LIN {X 0,Y 573.238,Z 117.075,A -85,B 0,C 180,E1 -2298.543,E2 -2298.543} C_VEL
LIN {X 0,Y 573.245,Z 117.077,A -85,B 0,C 180,E1 -2301.298,E2 -2301.298} C_VEL
LIN {X 0,Y 573.216,Z 117.081,A -85,B 0,C 180,E1 -2304.018,E2 -2304.018} C_VEL
LIN {X 0,Y 573.236,Z 117.074,A -85,B 0,C 180,E1 -2306.515,E2 -2306.515} C_VEL
LIN {X 0,Y 573.227,Z 117.08,A -85,B 0,C 180,E1 -2309.119,E2 -2309.119} C_VEL
LIN {X 0,Y 573.239,Z 117.083,A -85,B 0,C 180,E1 -2311.435,E2 -2311.435} C_VEL
LIN {X 0,Y 573.262,Z 117.073,A -85,B 0,C 180,E1 -2313.81,E2 -2313.81} C_VEL
LIN {X 0,Y 573.225,Z 117.076,A -85,B 0,C 180,E1 -2316.134,E2 -2316.134} C_VEL
LIN {X 0,Y 573.251,Z 117.082,A -85,B 0,C 180,E1 -2319.173,E2 -2319.173} C_VEL
LIN {X 0,Y 573.216,Z 117.081,A -85,B 0,C 180,E1 -2321.411,E2 -2321.411} C_VEL
LIN {X 0,Y 573.241,Z 117.076,A -85,B 0,C 180,E1 -2323.621,E2 -2323.621} C_VEL
LIN {X 0,Y 573.225,Z 117.08,A -85,B 0,C 180,E1 -2326.529,E2 -2326.529} C_VEL
LIN {X 0,Y 573.266,Z 117.08,A -85,B 0,C 180,E1 -2328.745,E2 -2328.745} C_VEL
LIN {X 0,Y 573.254,Z 117.074,A -85,B 0,C 180,E1 -2331.54,E2 -2331.54} C_VEL
LIN {X 0,Y 573.297,Z 117.073,A -85,B 0,C 180,E1 -2334.372,E2 -2334.372} C_VEL
LIN {X 0,Y 573.312,Z 117.068,A -85,B 0,C 180,E1 -2337.892,E2 -2337.892} C_VEL
LIN {X 0,Y 573.327,Z 117.071,A -85,B 0,C 180,E1 -2340.702,E2 -2340.702} C_VEL
LIN {X 0,Y 573.292,Z 117.073,A -85,B 0,C 180,E1 -2342.81,E2 -2342.81} C_VEL
LIN {X 0,Y 573.283,Z 117.071,A -85,B 0,C 180,E1 -2345.628,E2 -2345.628} C_VEL
LIN {X 0,Y 573.286,Z 117.101,A -85,B 0,C 180,E1 -2347.44,E2 -2347.44} C_VEL
LIN {X 0,Y 573.266,Z 128.019,A -85,B 0,C 180,E1 -2349.526,E2 -2349.526} C_VEL
LIN {X 0,Y 573.274,Z 136.889,A -85,B 0,C 180,E1 -2351.234,E2 -2351.234} C_VEL
LIN {X 0,Y 574.077,Z 143.404,A -85,B 0,C 180,E1 -2351.338,E2 -2351.338} C_VEL
LIN {X 0,Y 573.866,Z 242.802,A -85,B 0,C 180,E1 -2352.6,E2 -2352.6} C_VEL
LIN {X 0,Y 573.817,Z 251.677,A -85,B 0,C 180,E1 -2352.79,E2 -2352.79} C_VEL
LIN {X 0,Y 573.465,Z 255.472,A -85,B 0,C 180,E1 -2352.888,E2 -2352.888} C_VEL
LIN {X 0,Y 572.606,Z 259.214,A -85,B 0,C 180,E1 -2352.981,E2 -2352.981} C_VEL
LIN {X 0,Y 570.29,Z 266.507,A -85,B 0,C 180,E1 -2353.197,E2 -2353.197} C_VEL
LIN {X 0,Y 567.328,Z 275.39,A -85,B 0,C 180,E1 -2353.521,E2 -2353.521} C_VEL
LIN {X 0,Y 566.577,Z 280.637,A -85,B 0,C 180,E1 -2353.781,E2 -2353.781} C_VEL
LIN {X 0,Y 566.434,Z 291.364,A -85,B 0,C 180,E1 -2354.446,E2 -2354.446} C_VEL
LIN {X 0,Y 566.348,Z 300.093,A -85,B 0,C 180,E1 -2355.105,E2 -2355.105} C_VEL
LIN {X 0,Y 566.23,Z 308.332,A -85,B 0,C 180,E1 -2355.846,E2 -2355.846} C_VEL
LIN {X 0,Y 566.121,Z 316.358,A -85,B 0,C 180,E1 -2356.711,E2 -2356.711} C_VEL
LIN {X 0,Y 566.04,Z 322.701,A -85,B 0,C 180,E1 -2357.523,E2 -2357.523} C_VEL
LIN {X 0,Y 565.989,Z 328.827,A -85,B 0,C 180,E1 -2358.459,E2 -2358.459} C_VEL
LIN {X 0,Y 565.967,Z 334.819,A -85,B 0,C 180,E1 -2359.589,E2 -2359.589} C_VEL
LIN {X 0,Y 565.892,Z 339.537,A -85,B 0,C 180,E1 -2360.729,E2 -2360.729} C_VEL
LIN {X 0,Y 565.862,Z 343.032,A -85,B 0,C 180,E1 -2361.876,E2 -2361.876} C_VEL
LIN {X 0,Y 565.832,Z 345.629,A -85,B 0,C 180,E1 -2363.201,E2 -2363.201} C_VEL
LIN {X 0,Y 565.826,Z 346.693,A -85,B 0,C 180,E1 -2364.197,E2 -2364.197} C_VEL
LIN {X 0,Y 565.827,Z 346.992,A -85,B 0,C 180,E1 -2364.98,E2 -2364.98} C_VEL
LIN {X 0,Y 565.831,Z 346.744,A -85,B 0,C 180,E1 -2365.767,E2 -2365.767} C_VEL
LIN {X 0,Y 565.858,Z 346.003,A -85,B 0,C 180,E1 -2366.588,E2 -2366.588} C_VEL
LIN {X 0,Y 565.84,Z 344.871,A -85,B 0,C 180,E1 -2367.358,E2 -2367.358} C_VEL
LIN {X 0,Y 565.896,Z 342.029,A -85,B 0,C 180,E1 -2368.564,E2 -2368.564} C_VEL
LIN {X 0,Y 565.917,Z 338.527,A -85,B 0,C 180,E1 -2369.621,E2 -2369.621} C_VEL
LIN {X 0,Y 565.956,Z 334.309,A -85,B 0,C 180,E1 -2370.606,E2 -2370.606} C_VEL
LIN {X 0,Y 566.026,Z 328.765,A -85,B 0,C 180,E1 -2371.64,E2 -2371.64} C_VEL
LIN {X 0,Y 566.05,Z 323.052,A -85,B 0,C 180,E1 -2372.518,E2 -2372.518} C_VEL
LIN {X 0,Y 566.128,Z 316.918,A -85,B 0,C 180,E1 -2373.313,E2 -2373.313} C_VEL
LIN {X 0,Y 566.211,Z 310.133,A -85,B 0,C 180,E1 -2374.063,E2 -2374.063} C_VEL
LIN {X 0,Y 566.305,Z 302.147,A -85,B 0,C 180,E1 -2374.811,E2 -2374.811} C_VEL
LIN {X 0,Y 566.42,Z 293.527,A -85,B 0,C 180,E1 -2375.489,E2 -2375.489} C_VEL
LIN {X 0,Y 566.549,Z 284.706,A -85,B 0,C 180,E1 -2376.068,E2 -2376.068} C_VEL
LIN {X 0,Y 566.641,Z 275.027,A -85,B 0,C 180,E1 -2376.592,E2 -2376.592} C_VEL
LIN {X 0,Y 566.744,Z 264.912,A -85,B 0,C 180,E1 -2377.028,E2 -2377.028} C_VEL
LIN {X 0,Y 566.798,Z 254.959,A -85,B 0,C 180,E1 -2377.358,E2 -2377.358} C_VEL
LIN {X 0,Y 566.919,Z 242.981,A -85,B 0,C 180,E1 -2377.642,E2 -2377.642} C_VEL
LIN {X 0,Y 567.001,Z 141.748,A -85,B 0,C 180,E1 -2378.948,E2 -2378.948} C_VEL
LIN {X 0,Y 566.194,Z 136.908,A -85,B 0,C 180,E1 -2379.039,E2 -2379.039} C_VEL
LIN {X 0,Y 566.356,Z 122.425,A -85,B 0,C 180,E1 -2381.879,E2 -2381.879} C_VEL
LIN {X 0,Y 566.244,Z 117.951,A -85,B 0,C 180,E1 -2382.791,E2 -2382.791} C_VEL
LIN {X 0,Y 566.199,Z 117.957,A -85,B 0,C 180,E1 -2386.048,E2 -2386.048} C_VEL
LIN {X 0,Y 566.179,Z 117.954,A -85,B 0,C 180,E1 -2388.861,E2 -2388.861} C_VEL
LIN {X 0,Y 566.186,Z 117.963,A -85,B 0,C 180,E1 -2391.637,E2 -2391.637} C_VEL
LIN {X 0,Y 566.161,Z 117.957,A -85,B 0,C 180,E1 -2394.308,E2 -2394.308} C_VEL
LIN {X 0,Y 566.204,Z 117.952,A -85,B 0,C 180,E1 -2396.896,E2 -2396.896} C_VEL
LIN {X 0,Y 566.175,Z 117.963,A -85,B 0,C 180,E1 -2399.407,E2 -2399.407} C_VEL
LIN {X 0,Y 566.211,Z 117.953,A -85,B 0,C 180,E1 -2401.857,E2 -2401.857} C_VEL
LIN {X 0,Y 566.212,Z 117.95,A -85,B 0,C 180,E1 -2404.251,E2 -2404.251} C_VEL
LIN {X 0,Y 566.171,Z 117.956,A -85,B 0,C 180,E1 -2406.718,E2 -2406.718} C_VEL
LIN {X 0,Y 566.207,Z 117.954,A -85,B 0,C 180,E1 -2409.662,E2 -2409.662} C_VEL
LIN {X 0,Y 566.197,Z 117.954,A -85,B 0,C 180,E1 -2412.668,E2 -2412.668} C_VEL
LIN {X 0,Y 566.234,Z 117.949,A -85,B 0,C 180,E1 -2415.627,E2 -2415.627} C_VEL
LIN {X 0,Y 566.234,Z 117.951,A -85,B 0,C 180,E1 -2418.675,E2 -2418.675} C_VEL
LIN {X 0,Y 566.226,Z 117.951,A -85,B 0,C 180,E1 -2421.434,E2 -2421.434} C_VEL
LIN {X 0,Y 566.264,Z 117.944,A -85,B 0,C 180,E1 -2424.301,E2 -2424.301} C_VEL
LIN {X 0,Y 566.284,Z 117.941,A -85,B 0,C 180,E1 -2427.866,E2 -2427.866} C_VEL
LIN {X 0,Y 566.305,Z 117.947,A -85,B 0,C 180,E1 -2430.711,E2 -2430.711} C_VEL
LIN {X 0,Y 566.271,Z 117.951,A -85,B 0,C 180,E1 -2432.845,E2 -2432.845} C_VEL
LIN {X 0,Y 566.262,Z 117.943,A -85,B 0,C 180,E1 -2435.698,E2 -2435.698} C_VEL
LIN {X 0,Y 566.233,Z 117.956,A -85,B 0,C 180,E1 -2438.565,E2 -2438.565} C_VEL
LIN {X 0,Y 566.24,Z 117.946,A -85,B 0,C 180,E1 -2441.454,E2 -2441.454} C_VEL
LIN {X 0,Y 566.233,Z 117.957,A -85,B 0,C 180,E1 -2444.506,E2 -2444.506} C_VEL
LIN {X 0,Y 566.197,Z 117.951,A -85,B 0,C 180,E1 -2447.331,E2 -2447.331} C_VEL
LIN {X 0,Y 566.212,Z 117.959,A -85,B 0,C 180,E1 -2450.337,E2 -2450.337} C_VEL
LIN {X 0,Y 566.167,Z 117.955,A -85,B 0,C 180,E1 -2453.281,E2 -2453.281} C_VEL
LIN {X 0,Y 566.212,Z 117.952,A -85,B 0,C 180,E1 -2455.749,E2 -2455.749} C_VEL
LIN {X 0,Y 566.2,Z 117.961,A -85,B 0,C 180,E1 -2458.202,E2 -2458.202} C_VEL
LIN {X 0,Y 566.191,Z 117.955,A -85,B 0,C 180,E1 -2460.592,E2 -2460.592} C_VEL
LIN {X 0,Y 566.226,Z 117.948,A -85,B 0,C 180,E1 -2463.101,E2 -2463.101} C_VEL
LIN {X 0,Y 566.212,Z 117.956,A -85,B 0,C 180,E1 -2466.216,E2 -2466.216} C_VEL
LIN {X 0,Y 566.22,Z 117.95,A -85,B 0,C 180,E1 -2469.273,E2 -2469.273} C_VEL
LIN {X 0,Y 566.211,Z 117.957,A -85,B 0,C 180,E1 -2472.087,E2 -2472.087} C_VEL
LIN {X 0,Y 566.17,Z 117.955,A -85,B 0,C 180,E1 -2475.036,E2 -2475.036} C_VEL
LIN {X 0,Y 566.215,Z 117.953,A -85,B 0,C 180,E1 -2478.136,E2 -2478.136} C_VEL
LIN {X 0,Y 566.219,Z 117.949,A -85,B 0,C 180,E1 -2480.727,E2 -2480.727} C_VEL
LIN {X 0,Y 566.181,Z 117.961,A -85,B 0,C 180,E1 -2483.788,E2 -2483.788} C_VEL
LIN {X 0,Y 566.208,Z 117.951,A -85,B 0,C 180,E1 -2486.266,E2 -2486.266} C_VEL
LIN {X 0,Y 566.196,Z 117.953,A -85,B 0,C 180,E1 -2488.922,E2 -2488.922} C_VEL
LIN {X 0,Y 566.208,Z 117.954,A -85,B 0,C 180,E1 -2491.858,E2 -2491.858} C_VEL
LIN {X 0,Y 566.211,Z 117.95,A -85,B 0,C 180,E1 -2494.251,E2 -2494.251} C_VEL
LIN {X 0,Y 566.17,Z 117.956,A -85,B 0,C 180,E1 -2496.718,E2 -2496.718} C_VEL
LIN {X 0,Y 566.211,Z 117.954,A -85,B 0,C 180,E1 -2499.663,E2 -2499.663} C_VEL
LIN {X 0,Y 566.197,Z 117.953,A -85,B 0,C 180,E1 -2502.669,E2 -2502.669} C_VEL
LIN {X 0,Y 566.232,Z 117.95,A -85,B 0,C 180,E1 -2505.627,E2 -2505.627} C_VEL
LIN {X 0,Y 566.233,Z 117.95,A -85,B 0,C 180,E1 -2508.675,E2 -2508.675} C_VEL
LIN {X 0,Y 566.226,Z 117.952,A -85,B 0,C 180,E1 -2511.435,E2 -2511.435} C_VEL
LIN {X 0,Y 566.264,Z 117.944,A -85,B 0,C 180,E1 -2514.302,E2 -2514.302} C_VEL
LIN {X 0,Y 566.284,Z 117.941,A -85,B 0,C 180,E1 -2517.867,E2 -2517.867} C_VEL
LIN {X 0,Y 566.303,Z 117.946,A -85,B 0,C 180,E1 -2520.711,E2 -2520.711} C_VEL
LIN {X 0,Y 566.269,Z 117.952,A -85,B 0,C 180,E1 -2522.846,E2 -2522.846} C_VEL
LIN {X 0,Y 566.264,Z 117.943,A -85,B 0,C 180,E1 -2525.699,E2 -2525.699} C_VEL
LIN {X 0,Y 566.232,Z 117.955,A -85,B 0,C 180,E1 -2528.566,E2 -2528.566} C_VEL
LIN {X 0,Y 566.241,Z 117.946,A -85,B 0,C 180,E1 -2531.455,E2 -2531.455} C_VEL
LIN {X 0,Y 566.233,Z 117.956,A -85,B 0,C 180,E1 -2534.507,E2 -2534.507} C_VEL
LIN {X 0,Y 566.199,Z 117.951,A -85,B 0,C 180,E1 -2537.332,E2 -2537.332} C_VEL
LIN {X 0,Y 566.213,Z 117.958,A -85,B 0,C 180,E1 -2540.337,E2 -2540.337} C_VEL
LIN {X 0,Y 566.168,Z 117.955,A -85,B 0,C 180,E1 -2543.281,E2 -2543.281} C_VEL
LIN {X 0,Y 566.214,Z 117.951,A -85,B 0,C 180,E1 -2545.749,E2 -2545.749} C_VEL
LIN {X 0,Y 566.202,Z 117.96,A -85,B 0,C 180,E1 -2548.202,E2 -2548.202} C_VEL
LIN {X 0,Y 566.19,Z 117.952,A -85,B 0,C 180,E1 -2551.077,E2 -2551.077} C_VEL
LIN {X 0,Y 566.211,Z 117.953,A -85,B 0,C 180,E1 -2553.734,E2 -2553.734} C_VEL
LIN {X 0,Y 566.199,Z 117.954,A -85,B 0,C 180,E1 -2556.57,E2 -2556.57} C_VEL
LIN {X 0,Y 566.222,Z 117.949,A -85,B 0,C 180,E1 -2559.273,E2 -2559.273} C_VEL
LIN {X 0,Y 566.214,Z 117.957,A -85,B 0,C 180,E1 -2562.088,E2 -2562.088} C_VEL
LIN {X 0,Y 566.174,Z 117.954,A -85,B 0,C 180,E1 -2565.036,E2 -2565.036} C_VEL
LIN {X 0,Y 566.213,Z 117.954,A -85,B 0,C 180,E1 -2568.137,E2 -2568.137} C_VEL
LIN {X 0,Y 566.222,Z 117.948,A -85,B 0,C 180,E1 -2570.727,E2 -2570.727} C_VEL
LIN {X 0,Y 566.185,Z 117.962,A -85,B 0,C 180,E1 -2573.789,E2 -2573.789} C_VEL
LIN {X 0,Y 566.213,Z 117.951,A -85,B 0,C 180,E1 -2576.266,E2 -2576.266} C_VEL
LIN {X 0,Y 566.192,Z 117.954,A -85,B 0,C 180,E1 -2578.924,E2 -2578.924} C_VEL
LIN {X 0,Y 566.213,Z 117.955,A -85,B 0,C 180,E1 -2581.858,E2 -2581.858} C_VEL
LIN {X 0,Y 566.215,Z 117.953,A -85,B 0,C 180,E1 -2584.251,E2 -2584.251} C_VEL
LIN {X 0,Y 566.262,Z 118.049,A -85,B 0,C 180,E1 -2585.603,E2 -2585.603} C_VEL
LIN {X 0,Y 567.124,Z 122.581,A -85,B 0,C 180,E1 -2586.268,E2 -2586.268} C_VEL
LIN {X 0,Y 566.954,Z 140.918,A -85,B 0,C 180,E1 -2588.792,E2 -2588.792} C_VEL
LIN {X 0,Y 566.77,Z 162.759,A -85,B 0,C 180,E1 -2591.754,E2 -2591.754} C_VEL
LIN {X 0,Y 566.5,Z 183.521,A -85,B 0,C 180,E1 -2594.531,E2 -2594.531} C_VEL
LIN {X 0,Y 566.428,Z 194.357,A -85,B 0,C 180,E1 -2595.987,E2 -2595.987} C_VEL
LIN {X 0,Y 567.151,Z 200.531,A -85,B 0,C 180,E1 -2596.086,E2 -2596.086} C_VEL
LIN {X 0,Y 566.963,Z 302.961,A -85,B 0,C 180,E1 -2597.403,E2 -2597.403} C_VEL
LIN {X 0,Y 566.838,Z 316.227,A -85,B 0,C 180,E1 -2597.719,E2 -2597.719} C_VEL
LIN {X 0,Y 566.739,Z 328.385,A -85,B 0,C 180,E1 -2598.148,E2 -2598.148} C_VEL
LIN {X 0,Y 566.603,Z 339.362,A -85,B 0,C 180,E1 -2598.666,E2 -2598.666} C_VEL
LIN {X 0,Y 566.466,Z 350.908,A -85,B 0,C 180,E1 -2599.365,E2 -2599.365} C_VEL
LIN {X 0,Y 566.336,Z 361.541,A -85,B 0,C 180,E1 -2600.176,E2 -2600.176} C_VEL
LIN {X 0,Y 566.207,Z 371.116,A -85,B 0,C 180,E1 -2601.074,E2 -2601.074} C_VEL
LIN {X 0,Y 566.112,Z 378.963,A -85,B 0,C 180,E1 -2601.972,E2 -2601.972} C_VEL
LIN {X 0,Y 566.003,Z 386.624,A -85,B 0,C 180,E1 -2603.047,E2 -2603.047} C_VEL
LIN {X 0,Y 566.004,Z 393.681,A -85,B 0,C 180,E1 -2604.299,E2 -2604.299} C_VEL
LIN {X 0,Y 565.933,Z 398.374,A -85,B 0,C 180,E1 -2605.37,E2 -2605.37} C_VEL
LIN {X 0,Y 565.927,Z 401.959,A -85,B 0,C 180,E1 -2606.44,E2 -2606.44} C_VEL
LIN {X 0,Y 565.878,Z 403.808,A -85,B 0,C 180,E1 -2607.153,E2 -2607.153} C_VEL
LIN {X 0,Y 565.846,Z 406.184,A -85,B 0,C 180,E1 -2608.577,E2 -2608.577} C_VEL
LIN {X 0,Y 565.839,Z 407,A -85,B 0,C 180,E1 -2610,E2 -2610} C_VEL
LIN {X 0,Y 565.846,Z 406.185,A -85,B 0,C 180,E1 -2611.424,E2 -2611.424} C_VEL
LIN {X 0,Y 565.878,Z 403.809,A -85,B 0,C 180,E1 -2612.848,E2 -2612.848} C_VEL
LIN {X 0,Y 565.926,Z 400.895,A -85,B 0,C 180,E1 -2613.917,E2 -2613.917} C_VEL
LIN {X 0,Y 565.878,Z 396.947,A -85,B 0,C 180,E1 -2614.988,E2 -2614.988} C_VEL
LIN {X 0,Y 566.002,Z 391.866,A -85,B 0,C 180,E1 -2616.059,E2 -2616.059} C_VEL
LIN {X 0,Y 566.041,Z 385.465,A -85,B 0,C 180,E1 -2617.133,E2 -2617.133} C_VEL
LIN {X 0,Y 566.134,Z 377.475,A -85,B 0,C 180,E1 -2618.208,E2 -2618.208} C_VEL
LIN {X 0,Y 566.229,Z 369.331,A -85,B 0,C 180,E1 -2619.106,E2 -2619.106} C_VEL
LIN {X 0,Y 566.348,Z 359.395,A -85,B 0,C 180,E1 -2620.005,E2 -2620.005} C_VEL
LIN {X 0,Y 566.536,Z 348.287,A -85,B 0,C 180,E1 -2620.807,E2 -2620.807} C_VEL
LIN {X 0,Y 566.613,Z 337.168,A -85,B 0,C 180,E1 -2621.447,E2 -2621.447} C_VEL
LIN {X 0,Y 566.777,Z 324.972,A -85,B 0,C 180,E1 -2621.988,E2 -2621.988} C_VEL
LIN {X 0,Y 566.918,Z 312.164,A -85,B 0,C 180,E1 -2622.394,E2 -2622.394} C_VEL
LIN {X 0,Y 566.994,Z 300.087,A -85,B 0,C 180,E1 -2622.642,E2 -2622.642} C_VEL
LIN {X 0,Y 567.039,Z 198.7,A -85,B 0,C 180,E1 -2623.941,E2 -2623.941} C_VEL
LIN {X 0,Y 566.429,Z 194.268,A -85,B 0,C 180,E1 -2624.025,E2 -2624.025} C_VEL
LIN {X 0,Y 566.621,Z 172.686,A -85,B 0,C 180,E1 -2626.902,E2 -2626.902} C_VEL
LIN {X 0,Y 566.74,Z 153.686,A -85,B 0,C 180,E1 -2629.428,E2 -2629.428} C_VEL
LIN {X 0,Y 566.977,Z 132.946,A -85,B 0,C 180,E1 -2632.214,E2 -2632.214} C_VEL
LIN {X 0,Y 566.87,Z 121.427,A -85,B 0,C 180,E1 -2633.768,E2 -2633.768} C_VEL
LIN {X 0,Y 566.253,Z 117.954,A -85,B 0,C 180,E1 -2634.276,E2 -2634.276} C_VEL
LIN {X 0,Y 566.212,Z 117.952,A -85,B 0,C 180,E1 -2637.339,E2 -2637.339} C_VEL
LIN {X 0,Y 566.205,Z 117.955,A -85,B 0,C 180,E1 -2639.769,E2 -2639.769} C_VEL
LIN {X 0,Y 566.208,Z 117.958,A -85,B 0,C 180,E1 -2642.43,E2 -2642.43} C_VEL
LIN {X 0,Y 566.183,Z 117.955,A -85,B 0,C 180,E1 -2644.989,E2 -2644.989} C_VEL
LIN {X 0,Y 566.2,Z 117.953,A -85,B 0,C 180,E1 -2647.461,E2 -2647.461} C_VEL
LIN {X 0,Y 566.211,Z 117.958,A -85,B 0,C 180,E1 -2650.199,E2 -2650.199} C_VEL
LIN {X 0,Y 566.205,Z 117.951,A -85,B 0,C 180,E1 -2653.054,E2 -2653.054} C_VEL
LIN {X 0,Y 566.203,Z 117.958,A -85,B 0,C 180,E1 -2656.049,E2 -2656.049} C_VEL
LIN {X 0,Y 566.18,Z 117.953,A -85,B 0,C 180,E1 -2658.861,E2 -2658.861} C_VEL
LIN {X 0,Y 566.189,Z 117.961,A -85,B 0,C 180,E1 -2661.637,E2 -2661.637} C_VEL
LIN {X 0,Y 566.165,Z 117.956,A -85,B 0,C 180,E1 -2664.308,E2 -2664.308} C_VEL
LIN {X 0,Y 566.204,Z 117.952,A -85,B 0,C 180,E1 -2666.896,E2 -2666.896} C_VEL
LIN {X 0,Y 566.178,Z 117.962,A -85,B 0,C 180,E1 -2669.407,E2 -2669.407} C_VEL
LIN {X 0,Y 566.198,Z 117.954,A -85,B 0,C 180,E1 -2671.856,E2 -2671.856} C_VEL
LIN {X 0,Y 566.212,Z 117.949,A -85,B 0,C 180,E1 -2674.251,E2 -2674.251} C_VEL
LIN {X 0,Y 566.171,Z 117.958,A -85,B 0,C 180,E1 -2676.719,E2 -2676.719} C_VEL
LIN {X 0,Y 566.208,Z 117.952,A -85,B 0,C 180,E1 -2679.662,E2 -2679.662} C_VEL
LIN {X 0,Y 566.191,Z 117.956,A -85,B 0,C 180,E1 -2682.668,E2 -2682.668} C_VEL
LIN {X 0,Y 566.218,Z 117.95,A -85,B 0,C 180,E1 -2685.626,E2 -2685.626} C_VEL
LIN {X 0,Y 566.238,Z 117.954,A -85,B 0,C 180,E1 -2688.675,E2 -2688.675} C_VEL
LIN {X 0,Y 566.205,Z 117.953,A -85,B 0,C 180,E1 -2691.434,E2 -2691.434} C_VEL
LIN {X 0,Y 566.264,Z 117.949,A -85,B 0,C 180,E1 -2694.301,E2 -2694.301} C_VEL
LIN {X 0,Y 566.283,Z 117.943,A -85,B 0,C 180,E1 -2697.866,E2 -2697.866} C_VEL
LIN {X 0,Y 566.298,Z 117.946,A -85,B 0,C 180,E1 -2700.711,E2 -2700.711} C_VEL
LIN {X 0,Y 566.258,Z 117.949,A -85,B 0,C 180,E1 -2702.845,E2 -2702.845} C_VEL
LIN {X 0,Y 566.253,Z 117.948,A -85,B 0,C 180,E1 -2705.698,E2 -2705.698} C_VEL
LIN {X 0,Y 566.252,Z 118.121,A -85,B 0,C 180,E1 -2707.443,E2 -2707.443} C_VEL
LIN {X 0,Y 566.2,Z 131.558,A -85,B 0,C 180,E1 -2710.007,E2 -2710.007} C_VEL
LIN {X 0,Y 566.213,Z 136.969,A -85,B 0,C 180,E1 -2711.059,E2 -2711.059} C_VEL
LIN {X 0,Y 567.2,Z 143.266,A -85,B 0,C 180,E1 -2711.167,E2 -2711.167} C_VEL
LIN {X 0,Y 566.959,Z 243.635,A -85,B 0,C 180,E1 -2712.46,E2 -2712.46} C_VEL
LIN {X 0,Y 566.824,Z 255.084,A -85,B 0,C 180,E1 -2712.736,E2 -2712.736} C_VEL
LIN {X 0,Y 566.748,Z 265.353,A -85,B 0,C 180,E1 -2713.08,E2 -2713.08} C_VEL
LIN {X 0,Y 566.658,Z 273.964,A -85,B 0,C 180,E1 -2713.447,E2 -2713.447} C_VEL
LIN {X 0,Y 566.577,Z 280.637,A -85,B 0,C 180,E1 -2713.781,E2 -2713.781} C_VEL
LIN {X 0,Y 565.835,Z 285.792,A -85,B 0,C 180,E1 -2714.068,E2 -2714.068} C_VEL
LIN {X 0,Y 562.874,Z 294.015,A -85,B 0,C 180,E1 -2714.551,E2 -2714.551} C_VEL
LIN {X 0,Y 559.928,Z 301.744,A -85,B 0,C 180,E1 -2715.107,E2 -2715.107} C_VEL
LIN {X 0,Y 559.21,Z 306.115,A -85,B 0,C 180,E1 -2715.506,E2 -2715.506} C_VEL
LIN {X 0,Y 559.104,Z 314.877,A -85,B 0,C 180,E1 -2716.429,E2 -2716.429} C_VEL
LIN {X 0,Y 559,Z 321.75,A -85,B 0,C 180,E1 -2717.294,E2 -2717.294} C_VEL
LIN {X 0,Y 558.949,Z 327.38,A -85,B 0,C 180,E1 -2718.131,E2 -2718.131} C_VEL
LIN {X 0,Y 558.906,Z 332.705,A -85,B 0,C 180,E1 -2719.083,E2 -2719.083} C_VEL
LIN {X 0,Y 558.878,Z 336.333,A -85,B 0,C 180,E1 -2719.848,E2 -2719.848} C_VEL
LIN {X 0,Y 558.829,Z 340.62,A -85,B 0,C 180,E1 -2721.003,E2 -2721.003} C_VEL
LIN {X 0,Y 558.76,Z 343.764,A -85,B 0,C 180,E1 -2722.168,E2 -2722.168} C_VEL
LIN {X 0,Y 558.724,Z 345.806,A -85,B 0,C 180,E1 -2723.329,E2 -2723.329} C_VEL
LIN {X 0,Y 558.721,Z 346.821,A -85,B 0,C 180,E1 -2724.525,E2 -2724.525} C_VEL
LIN {X 0,Y 558.736,Z 346.922,A -85,B 0,C 180,E1 -2725.319,E2 -2725.319} C_VEL
LIN {X 0,Y 558.737,Z 346.56,A -85,B 0,C 180,E1 -2726.119,E2 -2726.119} C_VEL
LIN {X 0,Y 558.75,Z 345.602,A -85,B 0,C 180,E1 -2726.924,E2 -2726.924} C_VEL
LIN {X 0,Y 558.79,Z 342.893,A -85,B 0,C 180,E1 -2728.309,E2 -2728.309} C_VEL
LIN {X 0,Y 558.856,Z 339.701,A -85,B 0,C 180,E1 -2729.37,E2 -2729.37} C_VEL
LIN {X 0,Y 558.884,Z 334.587,A -85,B 0,C 180,E1 -2730.616,E2 -2730.616} C_VEL
LIN {X 0,Y 558.9,Z 329.925,A -85,B 0,C 180,E1 -2731.525,E2 -2731.525} C_VEL
LIN {X 0,Y 558.974,Z 324.363,A -85,B 0,C 180,E1 -2732.424,E2 -2732.424} C_VEL
LIN {X 0,Y 559.074,Z 317.346,A -85,B 0,C 180,E1 -2733.365,E2 -2733.365} C_VEL
LIN {X 0,Y 559.171,Z 310.258,A -85,B 0,C 180,E1 -2734.163,E2 -2734.163} C_VEL
LIN {X 0,Y 559.292,Z 302.86,A -85,B 0,C 180,E1 -2734.872,E2 -2734.872} C_VEL
LIN {X 0,Y 559.406,Z 294.876,A -85,B 0,C 180,E1 -2735.524,E2 -2735.524} C_VEL
LIN {X 0,Y 559.531,Z 287.034,A -85,B 0,C 180,E1 -2736.07,E2 -2736.07} C_VEL
LIN {X 0,Y 559.628,Z 276.465,A -85,B 0,C 180,E1 -2736.67,E2 -2736.67} C_VEL
LIN {X 0,Y 559.766,Z 266.591,A -85,B 0,C 180,E1 -2737.116,E2 -2737.116} C_VEL
LIN {X 0,Y 559.866,Z 256.265,A -85,B 0,C 180,E1 -2737.476,E2 -2737.476} C_VEL
LIN {X 0,Y 559.995,Z 244.528,A -85,B 0,C 180,E1 -2737.77,E2 -2737.77} C_VEL
LIN {X 0,Y 560.164,Z 199.077,A -85,B 0,C 180,E1 -2738.378,E2 -2738.378} C_VEL
LIN {X 0,Y 560.132,Z 142.677,A -85,B 0,C 180,E1 -2739.109,E2 -2739.109} C_VEL
LIN {X 0,Y 559.206,Z 137.155,A -85,B 0,C 180,E1 -2739.218,E2 -2739.218} C_VEL
LIN {X 0,Y 559.341,Z 122.233,A -85,B 0,C 180,E1 -2742.156,E2 -2742.156} C_VEL
LIN {X 0,Y 559.185,Z 118.83,A -85,B 0,C 180,E1 -2742.855,E2 -2742.855} C_VEL
LIN {X 0,Y 559.153,Z 118.839,A -85,B 0,C 180,E1 -2745.76,E2 -2745.76} C_VEL
LIN {X 0,Y 559.184,Z 118.827,A -85,B 0,C 180,E1 -2748.231,E2 -2748.231} C_VEL
LIN {X 0,Y 559.175,Z 118.829,A -85,B 0,C 180,E1 -2751.191,E2 -2751.191} C_VEL
LIN {X 0,Y 559.139,Z 118.837,A -85,B 0,C 180,E1 -2753.789,E2 -2753.789} C_VEL
LIN {X 0,Y 559.147,Z 118.83,A -85,B 0,C 180,E1 -2756.424,E2 -2756.424} C_VEL
LIN {X 0,Y 559.152,Z 118.832,A -85,B 0,C 180,E1 -2758.98,E2 -2758.98} C_VEL
LIN {X 0,Y 559.168,Z 118.834,A -85,B 0,C 180,E1 -2761.619,E2 -2761.619} C_VEL
LIN {X 0,Y 559.18,Z 118.828,A -85,B 0,C 180,E1 -2763.903,E2 -2763.903} C_VEL
LIN {X 0,Y 559.141,Z 118.831,A -85,B 0,C 180,E1 -2766.571,E2 -2766.571} C_VEL
LIN {X 0,Y 559.176,Z 118.834,A -85,B 0,C 180,E1 -2769.395,E2 -2769.395} C_VEL
LIN {X 0,Y 559.139,Z 118.833,A -85,B 0,C 180,E1 -2771.685,E2 -2771.685} C_VEL
LIN {X 0,Y 559.163,Z 118.828,A -85,B 0,C 180,E1 -2773.948,E2 -2773.948} C_VEL
LIN {X 0,Y 559.171,Z 118.827,A -85,B 0,C 180,E1 -2776.184,E2 -2776.184} C_VEL
LIN {X 0,Y 559.194,Z 118.832,A -85,B 0,C 180,E1 -2779.133,E2 -2779.133} C_VEL
LIN {X 0,Y 559.203,Z 118.823,A -85,B 0,C 180,E1 -2782.053,E2 -2782.053} C_VEL
LIN {X 0,Y 559.251,Z 118.826,A -85,B 0,C 180,E1 -2784.953,E2 -2784.953} C_VEL
LIN {X 0,Y 559.255,Z 118.816,A -85,B 0,C 180,E1 -2787.839,E2 -2787.839} C_VEL
LIN {X 0,Y 559.274,Z 118.822,A -85,B 0,C 180,E1 -2790.72,E2 -2790.72} C_VEL
LIN {X 0,Y 559.237,Z 118.826,A -85,B 0,C 180,E1 -2792.881,E2 -2792.881} C_VEL
LIN {X 0,Y 559.231,Z 118.819,A -85,B 0,C 180,E1 -2795.77,E2 -2795.77} C_VEL
LIN {X 0,Y 559.191,Z 118.833,A -85,B 0,C 180,E1 -2798.674,E2 -2798.674} C_VEL
LIN {X 0,Y 559.203,Z 118.823,A -85,B 0,C 180,E1 -2801.6,E2 -2801.6} C_VEL
LIN {X 0,Y 559.198,Z 118.832,A -85,B 0,C 180,E1 -2804.595,E2 -2804.595} C_VEL
LIN {X 0,Y 559.157,Z 118.829,A -85,B 0,C 180,E1 -2807.557,E2 -2807.557} C_VEL
LIN {X 0,Y 559.17,Z 118.829,A -85,B 0,C 180,E1 -2809.837,E2 -2809.837} C_VEL
LIN {X 0,Y 559.139,Z 118.837,A -85,B 0,C 180,E1 -2812.153,E2 -2812.153} C_VEL
LIN {X 0,Y 559.174,Z 118.826,A -85,B 0,C 180,E1 -2815.298,E2 -2815.298} C_VEL
LIN {X 0,Y 559.154,Z 118.831,A -85,B 0,C 180,E1 -2817.713,E2 -2817.713} C_VEL
LIN {X 0,Y 559.166,Z 118.837,A -85,B 0,C 180,E1 -2820.182,E2 -2820.182} C_VEL
LIN {X 0,Y 559.173,Z 118.828,A -85,B 0,C 180,E1 -2822.714,E2 -2822.714} C_VEL
LIN {X 0,Y 559.144,Z 118.831,A -85,B 0,C 180,E1 -2825.322,E2 -2825.322} C_VEL
LIN {X 0,Y 559.133,Z 118.841,A -85,B 0,C 180,E1 -2828.017,E2 -2828.017} C_VEL
LIN {X 0,Y 559.174,Z 118.826,A -85,B 0,C 180,E1 -2830.81,E2 -2830.81} C_VEL
LIN {X 0,Y 559.16,Z 118.836,A -85,B 0,C 180,E1 -2833.732,E2 -2833.732} C_VEL
LIN {X 0,Y 559.144,Z 118.83,A -85,B 0,C 180,E1 -2836.803,E2 -2836.803} C_VEL
LIN {X 0,Y 559.174,Z 118.828,A -85,B 0,C 180,E1 -2839.19,E2 -2839.19} C_VEL
LIN {X 0,Y 559.132,Z 118.837,A -85,B 0,C 180,E1 -2841.983,E2 -2841.983} C_VEL
LIN {X 0,Y 559.129,Z 118.832,A -85,B 0,C 180,E1 -2844.787,E2 -2844.787} C_VEL
LIN {X 0,Y 559.172,Z 118.833,A -85,B 0,C 180,E1 -2847.361,E2 -2847.361} C_VEL
LIN {X 0,Y 559.146,Z 118.831,A -85,B 0,C 180,E1 -2850.142,E2 -2850.142} C_VEL
LIN {X 0,Y 559.167,Z 118.831,A -85,B 0,C 180,E1 -2853.098,E2 -2853.098} C_VEL
LIN {X 0,Y 559.154,Z 118.837,A -85,B 0,C 180,E1 -2855.495,E2 -2855.495} C_VEL
LIN {X 0,Y 559.169,Z 118.828,A -85,B 0,C 180,E1 -2858.624,E2 -2858.624} C_VEL
LIN {X 0,Y 559.166,Z 118.831,A -85,B 0,C 180,E1 -2860.926,E2 -2860.926} C_VEL
LIN {X 0,Y 559.163,Z 118.828,A -85,B 0,C 180,E1 -2863.948,E2 -2863.948} C_VEL
LIN {X 0,Y 559.17,Z 118.827,A -85,B 0,C 180,E1 -2866.184,E2 -2866.184} C_VEL
LIN {X 0,Y 559.193,Z 118.834,A -85,B 0,C 180,E1 -2869.134,E2 -2869.134} C_VEL
LIN {X 0,Y 559.202,Z 118.823,A -85,B 0,C 180,E1 -2872.054,E2 -2872.054} C_VEL
LIN {X 0,Y 559.251,Z 118.826,A -85,B 0,C 180,E1 -2874.954,E2 -2874.954} C_VEL
LIN {X 0,Y 559.254,Z 118.816,A -85,B 0,C 180,E1 -2877.84,E2 -2877.84} C_VEL
LIN {X 0,Y 559.273,Z 118.822,A -85,B 0,C 180,E1 -2880.72,E2 -2880.72} C_VEL
LIN {X 0,Y 559.236,Z 118.827,A -85,B 0,C 180,E1 -2882.882,E2 -2882.882} C_VEL
LIN {X 0,Y 559.234,Z 118.819,A -85,B 0,C 180,E1 -2885.77,E2 -2885.77} C_VEL
LIN {X 0,Y 559.191,Z 118.834,A -85,B 0,C 180,E1 -2888.675,E2 -2888.675} C_VEL
LIN {X 0,Y 559.204,Z 118.823,A -85,B 0,C 180,E1 -2891.601,E2 -2891.601} C_VEL
LIN {X 0,Y 559.199,Z 118.833,A -85,B 0,C 180,E1 -2894.596,E2 -2894.596} C_VEL
LIN {X 0,Y 559.158,Z 118.828,A -85,B 0,C 180,E1 -2897.557,E2 -2897.557} C_VEL
LIN {X 0,Y 559.172,Z 118.828,A -85,B 0,C 180,E1 -2899.838,E2 -2899.838} C_VEL
LIN {X 0,Y 559.141,Z 118.836,A -85,B 0,C 180,E1 -2902.153,E2 -2902.153} C_VEL
LIN {X 0,Y 559.175,Z 118.826,A -85,B 0,C 180,E1 -2905.298,E2 -2905.298} C_VEL
LIN {X 0,Y 559.156,Z 118.83,A -85,B 0,C 180,E1 -2907.714,E2 -2907.714} C_VEL
LIN {X 0,Y 559.153,Z 118.838,A -85,B 0,C 180,E1 -2910.183,E2 -2910.183} C_VEL
LIN {X 0,Y 559.156,Z 118.831,A -85,B 0,C 180,E1 -2912.716,E2 -2912.716} C_VEL
LIN {X 0,Y 559.127,Z 118.833,A -85,B 0,C 180,E1 -2915.324,E2 -2915.324} C_VEL
LIN {X 0,Y 559.135,Z 118.841,A -85,B 0,C 180,E1 -2918.018,E2 -2918.018} C_VEL
LIN {X 0,Y 559.177,Z 118.826,A -85,B 0,C 180,E1 -2920.811,E2 -2920.811} C_VEL
LIN {X 0,Y 559.142,Z 118.837,A -85,B 0,C 180,E1 -2923.734,E2 -2923.734} C_VEL
LIN {X 0,Y 559.147,Z 118.83,A -85,B 0,C 180,E1 -2926.804,E2 -2926.804} C_VEL
LIN {X 0,Y 559.177,Z 118.827,A -85,B 0,C 180,E1 -2929.19,E2 -2929.19} C_VEL
LIN {X 0,Y 559.136,Z 118.837,A -85,B 0,C 180,E1 -2931.983,E2 -2931.983} C_VEL
LIN {X 0,Y 559.132,Z 118.832,A -85,B 0,C 180,E1 -2934.788,E2 -2934.788} C_VEL
LIN {X 0,Y 559.158,Z 118.834,A -85,B 0,C 180,E1 -2937.365,E2 -2937.365} C_VEL
LIN {X 0,Y 559.15,Z 118.832,A -85,B 0,C 180,E1 -2940.143,E2 -2940.143} C_VEL
LIN {X 0,Y 559.171,Z 118.831,A -85,B 0,C 180,E1 -2943.098,E2 -2943.098} C_VEL
LIN {X 0,Y 559.221,Z 118.943,A -85,B 0,C 180,E1 -2945.449,E2 -2945.449} C_VEL
LIN {X 0,Y 560.209,Z 124.91,A -85,B 0,C 180,E1 -2946.331,E2 -2946.331} C_VEL
LIN {X 0,Y 559.953,Z 143.02,A -85,B 0,C 180,E1 -2948.848,E2 -2948.848} C_VEL
LIN {X 0,Y 559.739,Z 165.243,A -85,B 0,C 180,E1 -2951.895,E2 -2951.895} C_VEL
LIN {X 0,Y 559.438,Z 186.007,A -85,B 0,C 180,E1 -2954.704,E2 -2954.704} C_VEL
LIN {X 0,Y 559.418,Z 194.127,A -85,B 0,C 180,E1 -2955.796,E2 -2955.796} C_VEL
LIN {X 0,Y 560.265,Z 202.043,A -85,B 0,C 180,E1 -2955.934,E2 -2955.934} C_VEL
LIN {X 0,Y 560.036,Z 302.959,A -85,B 0,C 180,E1 -2957.245,E2 -2957.245} C_VEL
LIN {X 0,Y 559.899,Z 316.226,A -85,B 0,C 180,E1 -2957.564,E2 -2957.564} C_VEL
LIN {X 0,Y 559.766,Z 329.504,A -85,B 0,C 180,E1 -2958.045,E2 -2958.045} C_VEL
LIN {X 0,Y 559.606,Z 341.415,A -85,B 0,C 180,E1 -2958.638,E2 -2958.638} C_VEL
LIN {X 0,Y 559.426,Z 353.488,A -85,B 0,C 180,E1 -2959.413,E2 -2959.413} C_VEL
LIN {X 0,Y 559.296,Z 363.649,A -85,B 0,C 180,E1 -2960.234,E2 -2960.234} C_VEL
LIN {X 0,Y 559.134,Z 372.788,A -85,B 0,C 180,E1 -2961.143,E2 -2961.143} C_VEL
LIN {X 0,Y 559.009,Z 381.69,A -85,B 0,C 180,E1 -2962.233,E2 -2962.233} C_VEL
LIN {X 0,Y 558.925,Z 387.741,A -85,B 0,C 180,E1 -2963.14,E2 -2963.14} C_VEL
LIN {X 0,Y 558.936,Z 393.681,A -85,B 0,C 180,E1 -2964.227,E2 -2964.227} C_VEL
LIN {X 0,Y 558.826,Z 398.374,A -85,B 0,C 180,E1 -2965.311,E2 -2965.311} C_VEL
LIN {X 0,Y 558.836,Z 401.959,A -85,B 0,C 180,E1 -2966.395,E2 -2966.395} C_VEL
LIN {X 0,Y 558.799,Z 403.808,A -85,B 0,C 180,E1 -2967.117,E2 -2967.117} C_VEL
LIN {X 0,Y 558.745,Z 406.183,A -85,B 0,C 180,E1 -2968.559,E2 -2968.559} C_VEL
LIN {X 0,Y 558.74,Z 407,A -85,B 0,C 180,E1 -2970,E2 -2970} C_VEL
LIN {X 0,Y 558.745,Z 406.184,A -85,B 0,C 180,E1 -2971.442,E2 -2971.442} C_VEL
LIN {X 0,Y 558.799,Z 403.809,A -85,B 0,C 180,E1 -2972.884,E2 -2972.884} C_VEL
LIN {X 0,Y 558.844,Z 400.895,A -85,B 0,C 180,E1 -2973.966,E2 -2973.966} C_VEL
LIN {X 0,Y 558.798,Z 396.947,A -85,B 0,C 180,E1 -2975.051,E2 -2975.051} C_VEL
LIN {X 0,Y 558.922,Z 391.866,A -85,B 0,C 180,E1 -2976.136,E2 -2976.136} C_VEL
LIN {X 0,Y 558.978,Z 385.465,A -85,B 0,C 180,E1 -2977.223,E2 -2977.223} C_VEL
LIN {X 0,Y 559.099,Z 377.475,A -85,B 0,C 180,E1 -2978.312,E2 -2978.312} C_VEL
LIN {X 0,Y 559.195,Z 369.331,A -85,B 0,C 180,E1 -2979.221,E2 -2979.221} C_VEL
LIN {X 0,Y 559.357,Z 359.394,A -85,B 0,C 180,E1 -2980.131,E2 -2980.131} C_VEL
LIN {X 0,Y 559.556,Z 348.393,A -85,B 0,C 180,E1 -2980.937,E2 -2980.937} C_VEL
LIN {X 0,Y 559.672,Z 336.451,A -85,B 0,C 180,E1 -2981.628,E2 -2981.628} C_VEL
LIN {X 0,Y 559.821,Z 324.969,A -85,B 0,C 180,E1 -2982.139,E2 -2982.139} C_VEL
LIN {X 0,Y 559.996,Z 312.162,A -85,B 0,C 180,E1 -2982.549,E2 -2982.549} C_VEL
LIN {X 0,Y 560.079,Z 300.082,A -85,B 0,C 180,E1 -2982.801,E2 -2982.801} C_VEL
LIN {X 0,Y 560.224,Z 199.984,A -85,B 0,C 180,E1 -2984.092,E2 -2984.092} C_VEL
LIN {X 0,Y 559.393,Z 194.034,A -85,B 0,C 180,E1 -2984.205,E2 -2984.205} C_VEL
LIN {X 0,Y 559.633,Z 171.172,A -85,B 0,C 180,E1 -2987.255,E2 -2987.255} C_VEL
LIN {X 0,Y 559.836,Z 149.36,A -85,B 0,C 180,E1 -2990.196,E2 -2990.196} C_VEL
LIN {X 0,Y 560.031,Z 128.061,A -85,B 0,C 180,E1 -2993.09,E2 -2993.09} C_VEL
LIN {X 0,Y 559.851,Z 122.304,A -85,B 0,C 180,E1 -2993.882,E2 -2993.882} C_VEL
LIN {X 0,Y 559.209,Z 118.832,A -85,B 0,C 180,E1 -2994.404,E2 -2994.404} C_VEL
LIN {X 0,Y 559.173,Z 118.832,A -85,B 0,C 180,E1 -2996.902,E2 -2996.902} C_VEL
LIN {X 0,Y 559.152,Z 118.835,A -85,B 0,C 180,E1 -2999.857,E2 -2999.857} C_VEL
LIN {X 0,Y 559.161,Z 118.832,A -85,B 0,C 180,E1 -3002.715,E2 -3002.715} C_VEL
LIN {X 0,Y 559.131,Z 118.833,A -85,B 0,C 180,E1 -3005.324,E2 -3005.324} C_VEL
LIN {X 0,Y 559.138,Z 118.84,A -85,B 0,C 180,E1 -3008.017,E2 -3008.017} C_VEL
LIN {X 0,Y 559.159,Z 118.83,A -85,B 0,C 180,E1 -3010.812,E2 -3010.812} C_VEL
LIN {X 0,Y 559.145,Z 118.837,A -85,B 0,C 180,E1 -3013.734,E2 -3013.734} C_VEL
LIN {X 0,Y 559.15,Z 118.83,A -85,B 0,C 180,E1 -3016.803,E2 -3016.803} C_VEL
LIN {X 0,Y 559.16,Z 118.829,A -85,B 0,C 180,E1 -3019.188,E2 -3019.188} C_VEL
LIN {X 0,Y 559.136,Z 118.836,A -85,B 0,C 180,E1 -3021.982,E2 -3021.982} C_VEL
LIN {X 0,Y 559.134,Z 118.832,A -85,B 0,C 180,E1 -3024.787,E2 -3024.787} C_VEL
LIN {X 0,Y 559.157,Z 118.836,A -85,B 0,C 180,E1 -3027.365,E2 -3027.365} C_VEL
LIN {X 0,Y 559.148,Z 118.831,A -85,B 0,C 180,E1 -3030.143,E2 -3030.143} C_VEL
LIN {X 0,Y 559.172,Z 118.833,A -85,B 0,C 180,E1 -3033.097,E2 -3033.097} C_VEL
LIN {X 0,Y 559.157,Z 118.835,A -85,B 0,C 180,E1 -3035.495,E2 -3035.495} C_VEL
LIN {X 0,Y 559.175,Z 118.829,A -85,B 0,C 180,E1 -3038.624,E2 -3038.624} C_VEL
LIN {X 0,Y 559.163,Z 118.835,A -85,B 0,C 180,E1 -3040.926,E2 -3040.926} C_VEL
LIN {X 0,Y 559.158,Z 118.829,A -85,B 0,C 180,E1 -3043.947,E2 -3043.947} C_VEL
LIN {X 0,Y 559.161,Z 118.829,A -85,B 0,C 180,E1 -3046.184,E2 -3046.184} C_VEL
LIN {X 0,Y 559.209,Z 118.829,A -85,B 0,C 180,E1 -3048.605,E2 -3048.605} C_VEL
LIN {X 0,Y 559.17,Z 118.83,A -85,B 0,C 180,E1 -3051.325,E2 -3051.325} C_VEL
LIN {X 0,Y 559.232,Z 118.824,A -85,B 0,C 180,E1 -3054.23,E2 -3054.23} C_VEL
LIN {X 0,Y 559.254,Z 118.819,A -85,B 0,C 180,E1 -3057.839,E2 -3057.839} C_VEL
LIN {X 0,Y 559.268,Z 118.822,A -85,B 0,C 180,E1 -3060.72,E2 -3060.72} C_VEL
LIN {X 0,Y 559.224,Z 118.825,A -85,B 0,C 180,E1 -3062.881,E2 -3062.881} C_VEL
LIN {X 0,Y 559.223,Z 118.825,A -85,B 0,C 180,E1 -3065.77,E2 -3065.77} C_VEL
LIN {X 0,Y 559.233,Z 119.022,A -85,B 0,C 180,E1 -3067.401,E2 -3067.401} C_VEL
LIN {X 0,Y 559.186,Z 131.446,A -85,B 0,C 180,E1 -3069.768,E2 -3069.768} C_VEL
LIN {X 0,Y 559.221,Z 137.291,A -85,B 0,C 180,E1 -3070.88,E2 -3070.88} C_VEL
LIN {X 0,Y 560.312,Z 144.719,A -85,B 0,C 180,E1 -3071.011,E2 -3071.011} C_VEL
LIN {X 0,Y 560.03,Z 243.266,A -85,B 0,C 180,E1 -3072.297,E2 -3072.297} C_VEL
LIN {X 0,Y 559.917,Z 254.844,A -85,B 0,C 180,E1 -3072.573,E2 -3072.573} C_VEL
LIN {X 0,Y 559.8,Z 265.248,A -85,B 0,C 180,E1 -3072.922,E2 -3072.922} C_VEL
LIN {X 0,Y 559.701,Z 274.832,A -85,B 0,C 180,E1 -3073.34,E2 -3073.34} C_VEL
LIN {X 0,Y 559.565,Z 283.504,A -85,B 0,C 180,E1 -3073.806,E2 -3073.806} C_VEL
LIN {X 0,Y 559.441,Z 292.131,A -85,B 0,C 180,E1 -3074.365,E2 -3074.365} C_VEL
LIN {X 0,Y 559.315,Z 300.243,A -85,B 0,C 180,E1 -3074.992,E2 -3074.992} C_VEL
LIN {X 0,Y 559.21,Z 306.115,A -85,B 0,C 180,E1 -3075.506,E2 -3075.506} C_VEL
LIN {X 0,Y 558.5,Z 310.396,A -85,B 0,C 180,E1 -3075.926,E2 -3075.926} C_VEL
LIN {X 0,Y 556.873,Z 314.461,A -85,B 0,C 180,E1 -3076.34,E2 -3076.34} C_VEL
LIN {X 0,Y 552.616,Z 323.148,A -85,B 0,C 180,E1 -3077.364,E2 -3077.364} C_VEL
LIN {X 0,Y 551.9,Z 326.49,A -85,B 0,C 180,E1 -3077.863,E2 -3077.863} C_VEL
LIN {X 0,Y 551.832,Z 332.572,A -85,B 0,C 180,E1 -3078.951,E2 -3078.951} C_VEL
LIN {X 0,Y 551.791,Z 337.688,A -85,B 0,C 180,E1 -3080.114,E2 -3080.114} C_VEL
LIN {X 0,Y 551.749,Z 340.503,A -85,B 0,C 180,E1 -3080.895,E2 -3080.895} C_VEL
LIN {X 0,Y 551.699,Z 342.753,A -85,B 0,C 180,E1 -3081.68,E2 -3081.68} C_VEL
LIN {X 0,Y 551.657,Z 344.454,A -85,B 0,C 180,E1 -3082.469,E2 -3082.469} C_VEL
LIN {X 0,Y 551.627,Z 345.984,A -85,B 0,C 180,E1 -3083.463,E2 -3083.463} C_VEL
LIN {X 0,Y 551.608,Z 346.625,A -85,B 0,C 180,E1 -3084.061,E2 -3084.061} C_VEL
LIN {X 0,Y 551.639,Z 346.946,A -85,B 0,C 180,E1 -3085.236,E2 -3085.236} C_VEL
LIN {X 0,Y 551.652,Z 345.65,A -85,B 0,C 180,E1 -3086.9,E2 -3086.9} C_VEL
LIN {X 0,Y 551.696,Z 343.439,A -85,B 0,C 180,E1 -3088.121,E2 -3088.121} C_VEL
LIN {X 0,Y 551.765,Z 339.963,A -85,B 0,C 180,E1 -3089.366,E2 -3089.366} C_VEL
LIN {X 0,Y 551.795,Z 334.966,A -85,B 0,C 180,E1 -3090.628,E2 -3090.628} C_VEL
LIN {X 0,Y 551.877,Z 329.594,A -85,B 0,C 180,E1 -3091.689,E2 -3091.689} C_VEL
LIN {X 0,Y 551.936,Z 324.169,A -85,B 0,C 180,E1 -3092.572,E2 -3092.572} C_VEL
LIN {X 0,Y 552.038,Z 318.073,A -85,B 0,C 180,E1 -3093.409,E2 -3093.409} C_VEL
LIN {X 0,Y 552.176,Z 310.404,A -85,B 0,C 180,E1 -3094.29,E2 -3094.29} C_VEL
LIN {X 0,Y 552.298,Z 302.793,A -85,B 0,C 180,E1 -3095.028,E2 -3095.028} C_VEL
LIN {X 0,Y 552.428,Z 294.502,A -85,B 0,C 180,E1 -3095.705,E2 -3095.705} C_VEL
LIN {X 0,Y 552.611,Z 284.705,A -85,B 0,C 180,E1 -3096.368,E2 -3096.368} C_VEL
LIN {X 0,Y 552.738,Z 274.981,A -85,B 0,C 180,E1 -3096.902,E2 -3096.902} C_VEL
LIN {X 0,Y 552.88,Z 263.169,A -85,B 0,C 180,E1 -3097.411,E2 -3097.411} C_VEL
LIN {X 0,Y 553.046,Z 249.326,A -85,B 0,C 180,E1 -3097.826,E2 -3097.826} C_VEL
LIN {X 0,Y 553.158,Z 235.671,A -85,B 0,C 180,E1 -3098.067,E2 -3098.067} C_VEL
LIN {X 0,Y 553.29,Z 143.728,A -85,B 0,C 180,E1 -3099.273,E2 -3099.273} C_VEL
LIN {X 0,Y 552.23,Z 137.447,A -85,B 0,C 180,E1 -3099.392,E2 -3099.392} C_VEL
LIN {X 0,Y 552.352,Z 121.969,A -85,B 0,C 180,E1 -3102.44,E2 -3102.44} C_VEL
LIN {X 0,Y 552.161,Z 119.706,A -85,B 0,C 180,E1 -3102.918,E2 -3102.918} C_VEL
LIN {X 0,Y 552.098,Z 119.716,A -85,B 0,C 180,E1 -3105.562,E2 -3105.562} C_VEL
LIN {X 0,Y 552.13,Z 119.704,A -85,B 0,C 180,E1 -3108.555,E2 -3108.555} C_VEL
LIN {X 0,Y 552.117,Z 119.711,A -85,B 0,C 180,E1 -3111.411,E2 -3111.411} C_VEL
LIN {X 0,Y 552.085,Z 119.711,A -85,B 0,C 180,E1 -3114.156,E2 -3114.156} C_VEL
LIN {X 0,Y 552.107,Z 119.708,A -85,B 0,C 180,E1 -3116.813,E2 -3116.813} C_VEL
LIN {X 0,Y 552.099,Z 119.716,A -85,B 0,C 180,E1 -3119.39,E2 -3119.39} C_VEL
LIN {X 0,Y 552.109,Z 119.709,A -85,B 0,C 180,E1 -3121.901,E2 -3121.901} C_VEL
LIN {X 0,Y 552.155,Z 119.701,A -85,B 0,C 180,E1 -3124.649,E2 -3124.649} C_VEL
LIN {X 0,Y 552.092,Z 119.714,A -85,B 0,C 180,E1 -3127.549,E2 -3127.549} C_VEL
LIN {X 0,Y 552.144,Z 119.702,A -85,B 0,C 180,E1 -3130.375,E2 -3130.375} C_VEL
LIN {X 0,Y 552.154,Z 119.707,A -85,B 0,C 180,E1 -3132.977,E2 -3132.977} C_VEL
LIN {X 0,Y 552.135,Z 119.703,A -85,B 0,C 180,E1 -3136.004,E2 -3136.004} C_VEL
LIN {X 0,Y 552.162,Z 119.709,A -85,B 0,C 180,E1 -3138.993,E2 -3138.993} C_VEL
LIN {X 0,Y 552.157,Z 119.7,A -85,B 0,C 180,E1 -3141.951,E2 -3141.951} C_VEL
LIN {X 0,Y 552.227,Z 119.701,A -85,B 0,C 180,E1 -3144.889,E2 -3144.889} C_VEL
LIN {X 0,Y 552.226,Z 119.692,A -85,B 0,C 180,E1 -3147.812,E2 -3147.812} C_VEL
LIN {X 0,Y 552.244,Z 119.698,A -85,B 0,C 180,E1 -3150.729,E2 -3150.729} C_VEL
LIN {X 0,Y 552.203,Z 119.702,A -85,B 0,C 180,E1 -3152.918,E2 -3152.918} C_VEL
LIN {X 0,Y 552.201,Z 119.695,A -85,B 0,C 180,E1 -3155.844,E2 -3155.844} C_VEL
LIN {X 0,Y 552.161,Z 119.707,A -85,B 0,C 180,E1 -3158.785,E2 -3158.785} C_VEL
LIN {X 0,Y 552.161,Z 119.7,A -85,B 0,C 180,E1 -3161.75,E2 -3161.75} C_VEL
LIN {X 0,Y 552.135,Z 119.709,A -85,B 0,C 180,E1 -3164.748,E2 -3164.748} C_VEL
LIN {X 0,Y 552.108,Z 119.708,A -85,B 0,C 180,E1 -3167.788,E2 -3167.788} C_VEL
LIN {X 0,Y 552.129,Z 119.709,A -85,B 0,C 180,E1 -3170.101,E2 -3170.101} C_VEL
LIN {X 0,Y 552.09,Z 119.717,A -85,B 0,C 180,E1 -3172.451,E2 -3172.451} C_VEL
LIN {X 0,Y 552.153,Z 119.701,A -85,B 0,C 180,E1 -3175.35,E2 -3175.35} C_VEL
LIN {X 0,Y 552.107,Z 119.715,A -85,B 0,C 180,E1 -3178.098,E2 -3178.098} C_VEL
LIN {X 0,Y 552.111,Z 119.709,A -85,B 0,C 180,E1 -3180.608,E2 -3180.608} C_VEL
LIN {X 0,Y 552.12,Z 119.705,A -85,B 0,C 180,E1 -3183.185,E2 -3183.185} C_VEL
LIN {X 0,Y 552.105,Z 119.713,A -85,B 0,C 180,E1 -3185.842,E2 -3185.842} C_VEL
LIN {X 0,Y 552.123,Z 119.705,A -85,B 0,C 180,E1 -3189.062,E2 -3189.062} C_VEL
LIN {X 0,Y 552.137,Z 119.706,A -85,B 0,C 180,E1 -3191.444,E2 -3191.444} C_VEL
LIN {X 0,Y 552.094,Z 119.709,A -85,B 0,C 180,E1 -3194.532,E2 -3194.532} C_VEL
LIN {X 0,Y 552.128,Z 119.71,A -85,B 0,C 180,E1 -3197.584,E2 -3197.584} C_VEL
LIN {X 0,Y 552.131,Z 119.704,A -85,B 0,C 180,E1 -3200.473,E2 -3200.473} C_VEL
LIN {X 0,Y 552.103,Z 119.711,A -85,B 0,C 180,E1 -3203.317,E2 -3203.317} C_VEL
LIN {X 0,Y 552.124,Z 119.709,A -85,B 0,C 180,E1 -3205.939,E2 -3205.939} C_VEL
LIN {X 0,Y 552.116,Z 119.706,A -85,B 0,C 180,E1 -3208.541,E2 -3208.541} C_VEL
LIN {X 0,Y 552.121,Z 119.714,A -85,B 0,C 180,E1 -3211.438,E2 -3211.438} C_VEL
LIN {X 0,Y 552.127,Z 119.704,A -85,B 0,C 180,E1 -3214.356,E2 -3214.356} C_VEL
LIN {X 0,Y 552.096,Z 119.709,A -85,B 0,C 180,E1 -3216.758,E2 -3216.758} C_VEL
LIN {X 0,Y 552.118,Z 119.712,A -85,B 0,C 180,E1 -3219.12,E2 -3219.12} C_VEL
LIN {X 0,Y 552.123,Z 119.712,A -85,B 0,C 180,E1 -3221.445,E2 -3221.445} C_VEL
LIN {X 0,Y 552.113,Z 119.708,A -85,B 0,C 180,E1 -3223.737,E2 -3223.737} C_VEL
LIN {X 0,Y 552.133,Z 119.704,A -85,B 0,C 180,E1 -3226.005,E2 -3226.005} C_VEL
LIN {X 0,Y 552.161,Z 119.708,A -85,B 0,C 180,E1 -3228.994,E2 -3228.994} C_VEL
LIN {X 0,Y 552.156,Z 119.701,A -85,B 0,C 180,E1 -3231.952,E2 -3231.952} C_VEL
LIN {X 0,Y 552.227,Z 119.7,A -85,B 0,C 180,E1 -3234.889,E2 -3234.889} C_VEL
LIN {X 0,Y 552.225,Z 119.692,A -85,B 0,C 180,E1 -3237.812,E2 -3237.812} C_VEL
LIN {X 0,Y 552.243,Z 119.697,A -85,B 0,C 180,E1 -3240.729,E2 -3240.729} C_VEL
LIN {X 0,Y 552.202,Z 119.703,A -85,B 0,C 180,E1 -3242.918,E2 -3242.918} C_VEL
LIN {X 0,Y 552.205,Z 119.695,A -85,B 0,C 180,E1 -3245.844,E2 -3245.844} C_VEL
LIN {X 0,Y 552.161,Z 119.708,A -85,B 0,C 180,E1 -3248.786,E2 -3248.786} C_VEL
LIN {X 0,Y 552.162,Z 119.7,A -85,B 0,C 180,E1 -3251.751,E2 -3251.751} C_VEL
LIN {X 0,Y 552.135,Z 119.71,A -85,B 0,C 180,E1 -3254.749,E2 -3254.749} C_VEL
LIN {X 0,Y 552.11,Z 119.707,A -85,B 0,C 180,E1 -3257.789,E2 -3257.789} C_VEL
LIN {X 0,Y 552.13,Z 119.708,A -85,B 0,C 180,E1 -3260.101,E2 -3260.101} C_VEL
LIN {X 0,Y 552.091,Z 119.717,A -85,B 0,C 180,E1 -3262.451,E2 -3262.451} C_VEL
LIN {X 0,Y 552.155,Z 119.701,A -85,B 0,C 180,E1 -3265.351,E2 -3265.351} C_VEL
LIN {X 0,Y 552.109,Z 119.713,A -85,B 0,C 180,E1 -3268.099,E2 -3268.099} C_VEL
LIN {X 0,Y 552.102,Z 119.711,A -85,B 0,C 180,E1 -3270.61,E2 -3270.61} C_VEL
LIN {X 0,Y 552.115,Z 119.706,A -85,B 0,C 180,E1 -3273.186,E2 -3273.186} C_VEL
LIN {X 0,Y 552.085,Z 119.715,A -85,B 0,C 180,E1 -3275.844,E2 -3275.844} C_VEL
LIN {X 0,Y 552.126,Z 119.704,A -85,B 0,C 180,E1 -3279.062,E2 -3279.062} C_VEL
LIN {X 0,Y 552.14,Z 119.705,A -85,B 0,C 180,E1 -3281.444,E2 -3281.444} C_VEL
LIN {X 0,Y 552.096,Z 119.71,A -85,B 0,C 180,E1 -3284.532,E2 -3284.532} C_VEL
LIN {X 0,Y 552.132,Z 119.709,A -85,B 0,C 180,E1 -3287.585,E2 -3287.585} C_VEL
LIN {X 0,Y 552.133,Z 119.704,A -85,B 0,C 180,E1 -3290.473,E2 -3290.473} C_VEL
LIN {X 0,Y 552.107,Z 119.71,A -85,B 0,C 180,E1 -3293.317,E2 -3293.317} C_VEL
LIN {X 0,Y 552.128,Z 119.709,A -85,B 0,C 180,E1 -3295.94,E2 -3295.94} C_VEL
LIN {X 0,Y 552.121,Z 119.706,A -85,B 0,C 180,E1 -3298.541,E2 -3298.541} C_VEL
LIN {X 0,Y 552.126,Z 119.713,A -85,B 0,C 180,E1 -3301.438,E2 -3301.438} C_VEL
LIN {X 0,Y 552.132,Z 119.708,A -85,B 0,C 180,E1 -3304.356,E2 -3304.356} C_VEL
LIN {X 0,Y 552.212,Z 119.861,A -85,B 0,C 180,E1 -3305.292,E2 -3305.292} C_VEL
LIN {X 0,Y 553.286,Z 126.337,A -85,B 0,C 180,E1 -3306.268,E2 -3306.268} C_VEL
LIN {X 0,Y 553.003,Z 144.079,A -85,B 0,C 180,E1 -3308.765,E2 -3308.765} C_VEL
LIN {X 0,Y 552.742,Z 166.302,A -85,B 0,C 180,E1 -3311.85,E2 -3311.85} C_VEL
LIN {X 0,Y 552.419,Z 185.682,A -85,B 0,C 180,E1 -3314.505,E2 -3314.505} C_VEL
LIN {X 0,Y 552.392,Z 194.071,A -85,B 0,C 180,E1 -3315.635,E2 -3315.635} C_VEL
LIN {X 0,Y 553.359,Z 201.316,A -85,B 0,C 180,E1 -3315.755,E2 -3315.755} C_VEL
LIN {X 0,Y 553.133,Z 302.166,A -85,B 0,C 180,E1 -3317.083,E2 -3317.083} C_VEL
LIN {X 0,Y 552.968,Z 315.639,A -85,B 0,C 180,E1 -3317.406,E2 -3317.406} C_VEL
LIN {X 0,Y 552.785,Z 329.049,A -85,B 0,C 180,E1 -3317.891,E2 -3317.891} C_VEL
LIN {X 0,Y 552.613,Z 340.841,A -85,B 0,C 180,E1 -3318.477,E2 -3318.477} C_VEL
LIN {X 0,Y 552.439,Z 351.972,A -85,B 0,C 180,E1 -3319.185,E2 -3319.185} C_VEL
LIN {X 0,Y 552.274,Z 362.482,A -85,B 0,C 180,E1 -3320.016,E2 -3320.016} C_VEL
LIN {X 0,Y 552.126,Z 371.073,A -85,B 0,C 180,E1 -3320.845,E2 -3320.845} C_VEL
LIN {X 0,Y 552.013,Z 378.963,A -85,B 0,C 180,E1 -3321.765,E2 -3321.765} C_VEL
LIN {X 0,Y 551.889,Z 386.623,A -85,B 0,C 180,E1 -3322.868,E2 -3322.868} C_VEL
LIN {X 0,Y 551.867,Z 393.681,A -85,B 0,C 180,E1 -3324.153,E2 -3324.153} C_VEL
LIN {X 0,Y 551.725,Z 398.374,A -85,B 0,C 180,E1 -3325.251,E2 -3325.251} C_VEL
LIN {X 0,Y 551.75,Z 401.959,A -85,B 0,C 180,E1 -3326.349,E2 -3326.349} C_VEL
LIN {X 0,Y 551.723,Z 403.807,A -85,B 0,C 180,E1 -3327.08,E2 -3327.08} C_VEL
LIN {X 0,Y 551.645,Z 406.182,A -85,B 0,C 180,E1 -3328.54,E2 -3328.54} C_VEL
LIN {X 0,Y 551.64,Z 407,A -85,B 0,C 180,E1 -3330,E2 -3330} C_VEL
LIN {X 0,Y 551.645,Z 406.183,A -85,B 0,C 180,E1 -3331.46,E2 -3331.46} C_VEL
LIN {X 0,Y 551.724,Z 403.809,A -85,B 0,C 180,E1 -3332.921,E2 -3332.921} C_VEL
LIN {X 0,Y 551.764,Z 400.894,A -85,B 0,C 180,E1 -3334.017,E2 -3334.017} C_VEL
LIN {X 0,Y 551.724,Z 396.947,A -85,B 0,C 180,E1 -3335.116,E2 -3335.116} C_VEL
LIN {X 0,Y 551.803,Z 391.189,A -85,B 0,C 180,E1 -3336.341,E2 -3336.341} C_VEL
LIN {X 0,Y 551.927,Z 384.233,A -85,B 0,C 180,E1 -3337.5,E2 -3337.5} C_VEL
LIN {X 0,Y 552.082,Z 375.984,A -85,B 0,C 180,E1 -3338.603,E2 -3338.603} C_VEL
LIN {X 0,Y 552.201,Z 367.456,A -85,B 0,C 180,E1 -3339.524,E2 -3339.524} C_VEL
LIN {X 0,Y 552.394,Z 356.892,A -85,B 0,C 180,E1 -3340.446,E2 -3340.446} C_VEL
LIN {X 0,Y 552.556,Z 345.969,A -85,B 0,C 180,E1 -3341.215,E2 -3341.215} C_VEL
LIN {X 0,Y 552.724,Z 334.965,A -85,B 0,C 180,E1 -3341.832,E2 -3341.832} C_VEL
LIN {X 0,Y 552.882,Z 323.156,A -85,B 0,C 180,E1 -3342.34,E2 -3342.34} C_VEL
LIN {X 0,Y 553.054,Z 310.462,A -85,B 0,C 180,E1 -3342.733,E2 -3342.733} C_VEL
LIN {X 0,Y 553.159,Z 297.481,A -85,B 0,C 180,E1 -3342.987,E2 -3342.987} C_VEL
LIN {X 0,Y 553.215,Z 200.196,A -85,B 0,C 180,E1 -3344.258,E2 -3344.258} C_VEL
LIN {X 0,Y 552.345,Z 193.635,A -85,B 0,C 180,E1 -3344.379,E2 -3344.379} C_VEL
LIN {X 0,Y 552.614,Z 172.45,A -85,B 0,C 180,E1 -3347.238,E2 -3347.238} C_VEL
LIN {X 0,Y 552.834,Z 150.25,A -85,B 0,C 180,E1 -3350.269,E2 -3350.269} C_VEL
LIN {X 0,Y 553.079,Z 127.715,A -85,B 0,C 180,E1 -3353.362,E2 -3353.362} C_VEL
LIN {X 0,Y 552.826,Z 123.135,A -85,B 0,C 180,E1 -3354.005,E2 -3354.005} C_VEL
LIN {X 0,Y 552.183,Z 119.707,A -85,B 0,C 180,E1 -3354.535,E2 -3354.535} C_VEL
LIN {X 0,Y 552.133,Z 119.707,A -85,B 0,C 180,E1 -3357.274,E2 -3357.274} C_VEL
LIN {X 0,Y 552.121,Z 119.714,A -85,B 0,C 180,E1 -3360.051,E2 -3360.051} C_VEL
LIN {X 0,Y 552.119,Z 119.708,A -85,B 0,C 180,E1 -3362.846,E2 -3362.846} C_VEL
LIN {X 0,Y 552.08,Z 119.712,A -85,B 0,C 180,E1 -3365.44,E2 -3365.44} C_VEL
LIN {X 0,Y 552.101,Z 119.714,A -85,B 0,C 180,E1 -3367.886,E2 -3367.886} C_VEL
LIN {X 0,Y 552.113,Z 119.71,A -85,B 0,C 180,E1 -3370.481,E2 -3370.481} C_VEL
LIN {X 0,Y 552.123,Z 119.709,A -85,B 0,C 180,E1 -3373.485,E2 -3373.485} C_VEL
LIN {X 0,Y 552.11,Z 119.707,A -85,B 0,C 180,E1 -3376.576,E2 -3376.576} C_VEL
LIN {X 0,Y 552.113,Z 119.711,A -85,B 0,C 180,E1 -3379.519,E2 -3379.519} C_VEL
LIN {X 0,Y 552.096,Z 119.709,A -85,B 0,C 180,E1 -3382.336,E2 -3382.336} C_VEL
LIN {X 0,Y 552.085,Z 119.712,A -85,B 0,C 180,E1 -3385.051,E2 -3385.051} C_VEL
LIN {X 0,Y 552.117,Z 119.711,A -85,B 0,C 180,E1 -3387.681,E2 -3387.681} C_VEL
LIN {X 0,Y 552.111,Z 119.707,A -85,B 0,C 180,E1 -3390.235,E2 -3390.235} C_VEL
LIN {X 0,Y 552.14,Z 119.708,A -85,B 0,C 180,E1 -3393,E2 -3393} C_VEL
LIN {X 0,Y 552.116,Z 119.713,A -85,B 0,C 180,E1 -3395.161,E2 -3395.161} C_VEL
LIN {X 0,Y 552.129,Z 119.705,A -85,B 0,C 180,E1 -3398.337,E2 -3398.337} C_VEL
LIN {X 0,Y 552.153,Z 119.704,A -85,B 0,C 180,E1 -3400.674,E2 -3400.674} C_VEL
LIN {X 0,Y 552.107,Z 119.708,A -85,B 0,C 180,E1 -3403.737,E2 -3403.737} C_VEL
LIN {X 0,Y 552.125,Z 119.705,A -85,B 0,C 180,E1 -3406.004,E2 -3406.004} C_VEL
LIN {X 0,Y 552.163,Z 119.708,A -85,B 0,C 180,E1 -3408.993,E2 -3408.993} C_VEL
LIN {X 0,Y 552.151,Z 119.703,A -85,B 0,C 180,E1 -3411.951,E2 -3411.951} C_VEL
LIN {X 0,Y 552.224,Z 119.7,A -85,B 0,C 180,E1 -3414.889,E2 -3414.889} C_VEL
LIN {X 0,Y 552.225,Z 119.695,A -85,B 0,C 180,E1 -3417.812,E2 -3417.812} C_VEL
LIN {X 0,Y 552.239,Z 119.698,A -85,B 0,C 180,E1 -3420.729,E2 -3420.729} C_VEL
LIN {X 0,Y 552.191,Z 119.701,A -85,B 0,C 180,E1 -3422.918,E2 -3422.918} C_VEL
LIN {X 0,Y 552.193,Z 119.701,A -85,B 0,C 180,E1 -3425.844,E2 -3425.844} C_VEL
LIN {X 0,Y 552.174,Z 119.813,A -85,B 0,C 180,E1 -3427.335,E2 -3427.335} C_VEL
LIN {X 0,Y 552.189,Z 129.507,A -85,B 0,C 180,E1 -3429.154,E2 -3429.154} C_VEL
LIN {X 0,Y 552.22,Z 137.707,A -85,B 0,C 180,E1 -3430.704,E2 -3430.704} C_VEL
LIN {X 0,Y 553.451,Z 145.447,A -85,B 0,C 180,E1 -3430.841,E2 -3430.841} C_VEL
LIN {X 0,Y 553.104,Z 243.804,A -85,B 0,C 180,E1 -3432.147,E2 -3432.147} C_VEL
LIN {X 0,Y 552.959,Z 256.362,A -85,B 0,C 180,E1 -3432.456,E2 -3432.456} C_VEL
LIN {X 0,Y 552.874,Z 267.591,A -85,B 0,C 180,E1 -3432.853,E2 -3432.853} C_VEL
LIN {X 0,Y 552.684,Z 279.593,A -85,B 0,C 180,E1 -3433.419,E2 -3433.419} C_VEL
LIN {X 0,Y 552.44,Z 291.687,A -85,B 0,C 180,E1 -3434.173,E2 -3434.173} C_VEL
LIN {X 0,Y 552.319,Z 301.124,A -85,B 0,C 180,E1 -3434.913,E2 -3434.913} C_VEL
LIN {X 0,Y 552.168,Z 309.404,A -85,B 0,C 180,E1 -3435.692,E2 -3435.692} C_VEL
LIN {X 0,Y 552.067,Z 316.248,A -85,B 0,C 180,E1 -3436.454,E2 -3436.454} C_VEL
LIN {X 0,Y 551.942,Z 322.389,A -85,B 0,C 180,E1 -3437.255,E2 -3437.255} C_VEL
LIN {X 0,Y 551.9,Z 326.49,A -85,B 0,C 180,E1 -3437.863,E2 -3437.863} C_VEL
LIN {X 0,Y 551.187,Z 329.623,A -85,B 0,C 180,E1 -3438.382,E2 -3438.382} C_VEL
LIN {X 0,Y 548.245,Z 334.316,A -85,B 0,C 180,E1 -3439.242,E2 -3439.242} C_VEL
LIN {X 0,Y 545.337,Z 338.39,A -85,B 0,C 180,E1 -3440.141,E2 -3440.141} C_VEL
LIN {X 0,Y 544.678,Z 340.489,A -85,B 0,C 180,E1 -3440.716,E2 -3440.716} C_VEL
LIN {X 0,Y 544.605,Z 343.945,A -85,B 0,C 180,E1 -3441.977,E2 -3441.977} C_VEL
LIN {X 0,Y 544.562,Z 345.525,A -85,B 0,C 180,E1 -3442.778,E2 -3442.778} C_VEL
LIN {X 0,Y 544.549,Z 346.576,A -85,B 0,C 180,E1 -3443.604,E2 -3443.604} C_VEL
LIN {X 0,Y 544.526,Z 347.155,A -85,B 0,C 180,E1 -3444.394,E2 -3444.394} C_VEL
LIN {X 0,Y 544.566,Z 347.27,A -85,B 0,C 180,E1 -3445.391,E2 -3445.391} C_VEL
LIN {X 0,Y 544.557,Z 347.008,A -85,B 0,C 180,E1 -3446.027,E2 -3446.027} C_VEL
LIN {X 0,Y 544.587,Z 345.871,A -85,B 0,C 180,E1 -3447.069,E2 -3447.069} C_VEL
LIN {X 0,Y 544.629,Z 342.548,A -85,B 0,C 180,E1 -3448.659,E2 -3448.659} C_VEL
LIN {X 0,Y 544.662,Z 339.07,A -85,B 0,C 180,E1 -3449.768,E2 -3449.768} C_VEL
LIN {X 0,Y 544.721,Z 333.62,A -85,B 0,C 180,E1 -3451.069,E2 -3451.069} C_VEL
LIN {X 0,Y 544.858,Z 326.542,A -85,B 0,C 180,E1 -3452.364,E2 -3452.364} C_VEL
LIN {X 0,Y 545.011,Z 318.57,A -85,B 0,C 180,E1 -3453.495,E2 -3453.495} C_VEL
LIN {X 0,Y 545.172,Z 310.735,A -85,B 0,C 180,E1 -3454.407,E2 -3454.407} C_VEL
LIN {X 0,Y 545.277,Z 302.332,A -85,B 0,C 180,E1 -3455.224,E2 -3455.224} C_VEL
LIN {X 0,Y 545.466,Z 293.136,A -85,B 0,C 180,E1 -3455.965,E2 -3455.965} C_VEL
LIN {X 0,Y 545.689,Z 282.442,A -85,B 0,C 180,E1 -3456.667,E2 -3456.667} C_VEL
LIN {X 0,Y 545.903,Z 270.193,A -85,B 0,C 180,E1 -3457.292,E2 -3457.292} C_VEL
LIN {X 0,Y 546.011,Z 257.555,A -85,B 0,C 180,E1 -3457.763,E2 -3457.763} C_VEL
LIN {X 0,Y 546.151,Z 244.823,A -85,B 0,C 180,E1 -3458.088,E2 -3458.088} C_VEL
LIN {X 0,Y 546.399,Z 144.315,A -85,B 0,C 180,E1 -3459.453,E2 -3459.453} C_VEL
LIN {X 0,Y 545.225,Z 137.767,A -85,B 0,C 180,E1 -3459.579,E2 -3459.579} C_VEL
LIN {X 0,Y 545.34,Z 123.488,A -85,B 0,C 180,E1 -3462.396,E2 -3462.396} C_VEL
LIN {X 0,Y 545.132,Z 120.583,A -85,B 0,C 180,E1 -3462.995,E2 -3462.995} C_VEL
LIN {X 0,Y 545.067,Z 120.588,A -85,B 0,C 180,E1 -3466.224,E2 -3466.224} C_VEL
LIN {X 0,Y 545.086,Z 120.582,A -85,B 0,C 180,E1 -3468.886,E2 -3468.886} C_VEL
LIN {X 0,Y 545.052,Z 120.593,A -85,B 0,C 180,E1 -3471.762,E2 -3471.762} C_VEL
LIN {X 0,Y 545.035,Z 120.588,A -85,B 0,C 180,E1 -3474.531,E2 -3474.531} C_VEL
LIN {X 0,Y 545.065,Z 120.589,A -85,B 0,C 180,E1 -3477.211,E2 -3477.211} C_VEL
LIN {X 0,Y 545.06,Z 120.589,A -85,B 0,C 180,E1 -3479.81,E2 -3479.81} C_VEL
LIN {X 0,Y 545.08,Z 120.582,A -85,B 0,C 180,E1 -3482.343,E2 -3482.343} C_VEL
LIN {X 0,Y 545.117,Z 120.58,A -85,B 0,C 180,E1 -3484.82,E2 -3484.82} C_VEL
LIN {X 0,Y 545.038,Z 120.596,A -85,B 0,C 180,E1 -3487.242,E2 -3487.242} C_VEL
LIN {X 0,Y 545.116,Z 120.578,A -85,B 0,C 180,E1 -3490.414,E2 -3490.414} C_VEL
LIN {X 0,Y 545.071,Z 120.587,A -85,B 0,C 180,E1 -3493.521,E2 -3493.521} C_VEL
LIN {X 0,Y 545.094,Z 120.581,A -85,B 0,C 180,E1 -3495.82,E2 -3495.82} C_VEL
LIN {X 0,Y 545.117,Z 120.584,A -85,B 0,C 180,E1 -3498.849,E2 -3498.849} C_VEL
LIN {X 0,Y 545.127,Z 120.576,A -85,B 0,C 180,E1 -3501.847,E2 -3501.847} C_VEL
LIN {X 0,Y 545.203,Z 120.575,A -85,B 0,C 180,E1 -3504.823,E2 -3504.823} C_VEL
LIN {X 0,Y 545.197,Z 120.568,A -85,B 0,C 180,E1 -3507.783,E2 -3507.783} C_VEL
LIN {X 0,Y 545.214,Z 120.574,A -85,B 0,C 180,E1 -3510.738,E2 -3510.738} C_VEL
LIN {X 0,Y 545.17,Z 120.577,A -85,B 0,C 180,E1 -3512.956,E2 -3512.956} C_VEL
LIN {X 0,Y 545.171,Z 120.571,A -85,B 0,C 180,E1 -3515.919,E2 -3515.919} C_VEL
LIN {X 0,Y 545.12,Z 120.582,A -85,B 0,C 180,E1 -3518.9,E2 -3518.9} C_VEL
LIN {X 0,Y 545.133,Z 120.577,A -85,B 0,C 180,E1 -3521.904,E2 -3521.904} C_VEL
LIN {X 0,Y 545.084,Z 120.585,A -85,B 0,C 180,E1 -3524.943,E2 -3524.943} C_VEL
LIN {X 0,Y 545.076,Z 120.586,A -85,B 0,C 180,E1 -3528.026,E2 -3528.026} C_VEL
LIN {X 0,Y 545.093,Z 120.59,A -85,B 0,C 180,E1 -3530.372,E2 -3530.372} C_VEL
LIN {X 0,Y 545.077,Z 120.583,A -85,B 0,C 180,E1 -3533.559,E2 -3533.559} C_VEL
LIN {X 0,Y 545.078,Z 120.588,A -85,B 0,C 180,E1 -3536,E2 -3536} C_VEL
LIN {X 0,Y 545.089,Z 120.583,A -85,B 0,C 180,E1 -3538.748,E2 -3538.748} C_VEL
LIN {X 0,Y 545.076,Z 120.586,A -85,B 0,C 180,E1 -3541.682,E2 -3541.682} C_VEL
LIN {X 0,Y 545.074,Z 120.585,A -85,B 0,C 180,E1 -3544.563,E2 -3544.563} C_VEL
LIN {X 0,Y 545.037,Z 120.588,A -85,B 0,C 180,E1 -3547.304,E2 -3547.304} C_VEL
LIN {X 0,Y 545.073,Z 120.589,A -85,B 0,C 180,E1 -3550.142,E2 -3550.142} C_VEL
LIN {X 0,Y 545.084,Z 120.582,A -85,B 0,C 180,E1 -3553.106,E2 -3553.106} C_VEL
LIN {X 0,Y 545.064,Z 120.588,A -85,B 0,C 180,E1 -3556.224,E2 -3556.224} C_VEL
LIN {X 0,Y 545.098,Z 120.58,A -85,B 0,C 180,E1 -3558.887,E2 -3558.887} C_VEL
LIN {X 0,Y 545.052,Z 120.594,A -85,B 0,C 180,E1 -3561.763,E2 -3561.763} C_VEL
LIN {X 0,Y 545.033,Z 120.588,A -85,B 0,C 180,E1 -3564.532,E2 -3564.532} C_VEL
LIN {X 0,Y 545.079,Z 120.586,A -85,B 0,C 180,E1 -3567.213,E2 -3567.213} C_VEL
LIN {X 0,Y 545.063,Z 120.589,A -85,B 0,C 180,E1 -3569.811,E2 -3569.811} C_VEL
LIN {X 0,Y 545.086,Z 120.581,A -85,B 0,C 180,E1 -3572.344,E2 -3572.344} C_VEL
LIN {X 0,Y 545.115,Z 120.579,A -85,B 0,C 180,E1 -3574.821,E2 -3574.821} C_VEL
LIN {X 0,Y 545.036,Z 120.595,A -85,B 0,C 180,E1 -3577.243,E2 -3577.243} C_VEL
LIN {X 0,Y 545.118,Z 120.577,A -85,B 0,C 180,E1 -3580.415,E2 -3580.415} C_VEL
LIN {X 0,Y 545.07,Z 120.588,A -85,B 0,C 180,E1 -3583.521,E2 -3583.521} C_VEL
LIN {X 0,Y 545.093,Z 120.582,A -85,B 0,C 180,E1 -3585.82,E2 -3585.82} C_VEL
LIN {X 0,Y 545.116,Z 120.583,A -85,B 0,C 180,E1 -3588.85,E2 -3588.85} C_VEL
LIN {X 0,Y 545.126,Z 120.577,A -85,B 0,C 180,E1 -3591.847,E2 -3591.847} C_VEL
LIN {X 0,Y 545.203,Z 120.574,A -85,B 0,C 180,E1 -3594.823,E2 -3594.823} C_VEL
LIN {X 0,Y 545.197,Z 120.568,A -85,B 0,C 180,E1 -3597.784,E2 -3597.784} C_VEL
LIN {X 0,Y 545.213,Z 120.573,A -85,B 0,C 180,E1 -3600.739,E2 -3600.739} C_VEL
LIN {X 0,Y 545.169,Z 120.578,A -85,B 0,C 180,E1 -3602.956,E2 -3602.956} C_VEL
LIN {X 0,Y 545.177,Z 120.57,A -85,B 0,C 180,E1 -3605.92,E2 -3605.92} C_VEL
LIN {X 0,Y 545.12,Z 120.583,A -85,B 0,C 180,E1 -3608.9,E2 -3608.9} C_VEL
LIN {X 0,Y 545.134,Z 120.576,A -85,B 0,C 180,E1 -3611.904,E2 -3611.904} C_VEL
LIN {X 0,Y 545.085,Z 120.585,A -85,B 0,C 180,E1 -3614.944,E2 -3614.944} C_VEL
LIN {X 0,Y 545.078,Z 120.585,A -85,B 0,C 180,E1 -3618.026,E2 -3618.026} C_VEL
LIN {X 0,Y 545.095,Z 120.589,A -85,B 0,C 180,E1 -3620.372,E2 -3620.372} C_VEL
LIN {X 0,Y 545.078,Z 120.583,A -85,B 0,C 180,E1 -3623.56,E2 -3623.56} C_VEL
LIN {X 0,Y 545.079,Z 120.587,A -85,B 0,C 180,E1 -3626.001,E2 -3626.001} C_VEL
LIN {X 0,Y 545.088,Z 120.584,A -85,B 0,C 180,E1 -3628.749,E2 -3628.749} C_VEL
LIN {X 0,Y 545.057,Z 120.587,A -85,B 0,C 180,E1 -3631.679,E2 -3631.679} C_VEL
LIN {X 0,Y 545.062,Z 120.587,A -85,B 0,C 180,E1 -3634.565,E2 -3634.565} C_VEL
LIN {X 0,Y 545.036,Z 120.588,A -85,B 0,C 180,E1 -3637.304,E2 -3637.304} C_VEL
LIN {X 0,Y 545.093,Z 120.588,A -85,B 0,C 180,E1 -3640.141,E2 -3640.141} C_VEL
LIN {X 0,Y 545.079,Z 120.582,A -85,B 0,C 180,E1 -3643.107,E2 -3643.107} C_VEL
LIN {X 0,Y 545.068,Z 120.588,A -85,B 0,C 180,E1 -3646.225,E2 -3646.225} C_VEL
LIN {X 0,Y 545.097,Z 120.58,A -85,B 0,C 180,E1 -3648.887,E2 -3648.887} C_VEL
LIN {X 0,Y 545.056,Z 120.595,A -85,B 0,C 180,E1 -3651.763,E2 -3651.763} C_VEL
LIN {X 0,Y 545.037,Z 120.588,A -85,B 0,C 180,E1 -3654.532,E2 -3654.532} C_VEL
LIN {X 0,Y 545.07,Z 120.586,A -85,B 0,C 180,E1 -3657.212,E2 -3657.212} C_VEL
LIN {X 0,Y 545.065,Z 120.59,A -85,B 0,C 180,E1 -3659.811,E2 -3659.811} C_VEL
LIN {X 0,Y 545.083,Z 120.584,A -85,B 0,C 180,E1 -3662.344,E2 -3662.344} C_VEL
LIN {X 0,Y 545.173,Z 120.78,A -85,B 0,C 180,E1 -3665.129,E2 -3665.129} C_VEL
LIN {X 0,Y 546.366,Z 128.12,A -85,B 0,C 180,E1 -3666.251,E2 -3666.251} C_VEL
LIN {X 0,Y 546.003,Z 147.919,A -85,B 0,C 180,E1 -3669.073,E2 -3669.073} C_VEL
LIN {X 0,Y 545.7,Z 170.567,A -85,B 0,C 180,E1 -3672.25,E2 -3672.25} C_VEL
LIN {X 0,Y 545.371,Z 191.322,A -85,B 0,C 180,E1 -3675.128,E2 -3675.128} C_VEL
LIN {X 0,Y 545.351,Z 193.495,A -85,B 0,C 180,E1 -3675.429,E2 -3675.429} C_VEL
LIN {X 0,Y 546.492,Z 203.181,A -85,B 0,C 180,E1 -3675.606,E2 -3675.606} C_VEL
LIN {X 0,Y 546.184,Z 302.546,A -85,B 0,C 180,E1 -3676.94,E2 -3676.94} C_VEL
LIN {X 0,Y 545.996,Z 315.745,A -85,B 0,C 180,E1 -3677.266,E2 -3677.266} C_VEL
LIN {X 0,Y 545.805,Z 328.459,A -85,B 0,C 180,E1 -3677.734,E2 -3677.734} C_VEL
LIN {X 0,Y 545.589,Z 340.313,A -85,B 0,C 180,E1 -3678.327,E2 -3678.327} C_VEL
LIN {X 0,Y 545.418,Z 351.475,A -85,B 0,C 180,E1 -3679.044,E2 -3679.044} C_VEL
LIN {X 0,Y 545.225,Z 362.007,A -85,B 0,C 180,E1 -3679.885,E2 -3679.885} C_VEL
LIN {X 0,Y 545.085,Z 370.619,A -85,B 0,C 180,E1 -3680.726,E2 -3680.726} C_VEL
LIN {X 0,Y 544.947,Z 378.561,A -85,B 0,C 180,E1 -3681.658,E2 -3681.658} C_VEL
LIN {X 0,Y 544.824,Z 386.316,A -85,B 0,C 180,E1 -3682.775,E2 -3682.775} C_VEL
LIN {X 0,Y 544.777,Z 393.461,A -85,B 0,C 180,E1 -3684.076,E2 -3684.076} C_VEL
LIN {X 0,Y 544.628,Z 398.207,A -85,B 0,C 180,E1 -3685.189,E2 -3685.189} C_VEL
LIN {X 0,Y 544.669,Z 401.84,A -85,B 0,C 180,E1 -3686.301,E2 -3686.301} C_VEL
LIN {X 0,Y 544.65,Z 403.712,A -85,B 0,C 180,E1 -3687.042,E2 -3687.042} C_VEL
LIN {X 0,Y 544.546,Z 406.111,A -85,B 0,C 180,E1 -3688.521,E2 -3688.521} C_VEL
LIN {X 0,Y 544.542,Z 406.722,A -85,B 0,C 180,E1 -3689.261,E2 -3689.261} C_VEL
LIN {X 0,Y 544.541,Z 406.94,A -85,B 0,C 180,E1 -3690,E2 -3690} C_VEL
LIN {X 0,Y 544.542,Z 406.722,A -85,B 0,C 180,E1 -3690.74,E2 -3690.74} C_VEL
LIN {X 0,Y 544.572,Z 405.112,A -85,B 0,C 180,E1 -3692.219,E2 -3692.219} C_VEL
LIN {X 0,Y 544.65,Z 403.712,A -85,B 0,C 180,E1 -3692.959,E2 -3692.959} C_VEL
LIN {X 0,Y 544.684,Z 400.759,A -85,B 0,C 180,E1 -3694.07,E2 -3694.07} C_VEL
LIN {X 0,Y 544.654,Z 396.754,A -85,B 0,C 180,E1 -3695.183,E2 -3695.183} C_VEL
LIN {X 0,Y 544.708,Z 391.438,A -85,B 0,C 180,E1 -3696.328,E2 -3696.328} C_VEL
LIN {X 0,Y 544.837,Z 385.113,A -85,B 0,C 180,E1 -3697.412,E2 -3697.412} C_VEL
LIN {X 0,Y 544.968,Z 377.015,A -85,B 0,C 180,E1 -3698.529,E2 -3698.529} C_VEL
LIN {X 0,Y 545.114,Z 368.758,A -85,B 0,C 180,E1 -3699.462,E2 -3699.462} C_VEL
LIN {X 0,Y 545.341,Z 358.683,A -85,B 0,C 180,E1 -3700.395,E2 -3700.395} C_VEL
LIN {X 0,Y 545.51,Z 347.705,A -85,B 0,C 180,E1 -3701.209,E2 -3701.209} C_VEL
LIN {X 0,Y 545.681,Z 336.109,A -85,B 0,C 180,E1 -3701.892,E2 -3701.892} C_VEL
LIN {X 0,Y 545.899,Z 323.699,A -85,B 0,C 180,E1 -3702.453,E2 -3702.453} C_VEL
LIN {X 0,Y 546.088,Z 311.442,A -85,B 0,C 180,E1 -3702.851,E2 -3702.851} C_VEL
LIN {X 0,Y 546.22,Z 299.383,A -85,B 0,C 180,E1 -3703.107,E2 -3703.107} C_VEL
LIN {X 0,Y 546.381,Z 201.334,A -85,B 0,C 180,E1 -3704.417,E2 -3704.417} C_VEL
LIN {X 0,Y 545.272,Z 193.084,A -85,B 0,C 180,E1 -3704.582,E2 -3704.582} C_VEL
LIN {X 0,Y 545.567,Z 173.623,A -85,B 0,C 180,E1 -3707.235,E2 -3707.235} C_VEL
LIN {X 0,Y 545.849,Z 151.143,A -85,B 0,C 180,E1 -3710.343,E2 -3710.343} C_VEL
LIN {X 0,Y 546.12,Z 129.776,A -85,B 0,C 180,E1 -3713.311,E2 -3713.311} C_VEL
LIN {X 0,Y 545.829,Z 124.338,A -85,B 0,C 180,E1 -3714.088,E2 -3714.088} C_VEL
LIN {X 0,Y 545.139,Z 120.584,A -85,B 0,C 180,E1 -3714.67,E2 -3714.67} C_VEL
LIN {X 0,Y 545.084,Z 120.586,A -85,B 0,C 180,E1 -3717.656,E2 -3717.656} C_VEL
LIN {X 0,Y 545.081,Z 120.593,A -85,B 0,C 180,E1 -3720.246,E2 -3720.246} C_VEL
LIN {X 0,Y 545.083,Z 120.583,A -85,B 0,C 180,E1 -3723.062,E2 -3723.062} C_VEL
LIN {X 0,Y 545.037,Z 120.591,A -85,B 0,C 180,E1 -3725.673,E2 -3725.673} C_VEL
LIN {X 0,Y 545.058,Z 120.593,A -85,B 0,C 180,E1 -3728.237,E2 -3728.237} C_VEL
LIN {X 0,Y 545.085,Z 120.586,A -85,B 0,C 180,E1 -3730.473,E2 -3730.473} C_VEL
LIN {X 0,Y 545.082,Z 120.583,A -85,B 0,C 180,E1 -3733.107,E2 -3733.107} C_VEL
LIN {X 0,Y 545.071,Z 120.587,A -85,B 0,C 180,E1 -3736.224,E2 -3736.224} C_VEL
LIN {X 0,Y 545.086,Z 120.581,A -85,B 0,C 180,E1 -3738.885,E2 -3738.885} C_VEL
LIN {X 0,Y 545.056,Z 120.593,A -85,B 0,C 180,E1 -3741.763,E2 -3741.763} C_VEL
LIN {X 0,Y 545.039,Z 120.587,A -85,B 0,C 180,E1 -3744.531,E2 -3744.531} C_VEL
LIN {X 0,Y 545.068,Z 120.588,A -85,B 0,C 180,E1 -3747.211,E2 -3747.211} C_VEL
LIN {X 0,Y 545.064,Z 120.588,A -85,B 0,C 180,E1 -3749.81,E2 -3749.81} C_VEL
LIN {X 0,Y 545.081,Z 120.583,A -85,B 0,C 180,E1 -3752.343,E2 -3752.343} C_VEL
LIN {X 0,Y 545.109,Z 120.581,A -85,B 0,C 180,E1 -3754.82,E2 -3754.82} C_VEL
LIN {X 0,Y 545.039,Z 120.595,A -85,B 0,C 180,E1 -3757.242,E2 -3757.242} C_VEL
LIN {X 0,Y 545.119,Z 120.578,A -85,B 0,C 180,E1 -3760.415,E2 -3760.415} C_VEL
LIN {X 0,Y 545.058,Z 120.587,A -85,B 0,C 180,E1 -3763.52,E2 -3763.52} C_VEL
LIN {X 0,Y 545.087,Z 120.582,A -85,B 0,C 180,E1 -3765.819,E2 -3765.819} C_VEL
LIN {X 0,Y 545.12,Z 120.586,A -85,B 0,C 180,E1 -3768.849,E2 -3768.849} C_VEL
LIN {X 0,Y 545.099,Z 120.581,A -85,B 0,C 180,E1 -3771.846,E2 -3771.846} C_VEL
LIN {X 0,Y 545.2,Z 120.576,A -85,B 0,C 180,E1 -3774.823,E2 -3774.823} C_VEL
LIN {X 0,Y 545.196,Z 120.57,A -85,B 0,C 180,E1 -3777.783,E2 -3777.783} C_VEL
LIN {X 0,Y 545.209,Z 120.573,A -85,B 0,C 180,E1 -3780.738,E2 -3780.738} C_VEL
LIN {X 0,Y 545.157,Z 120.577,A -85,B 0,C 180,E1 -3782.956,E2 -3782.956} C_VEL
LIN {X 0,Y 545.165,Z 120.578,A -85,B 0,C 180,E1 -3785.919,E2 -3785.919} C_VEL
LIN {X 0,Y 545.143,Z 120.675,A -85,B 0,C 180,E1 -3787.267,E2 -3787.267} C_VEL
LIN {X 0,Y 545.184,Z 131.45,A -85,B 0,C 180,E1 -3789.273,E2 -3789.273} C_VEL
LIN {X 0,Y 545.22,Z 138.009,A -85,B 0,C 180,E1 -3790.514,E2 -3790.514} C_VEL
LIN {X 0,Y 546.569,Z 145.248,A -85,B 0,C 180,E1 -3790.651,E2 -3790.651} C_VEL
LIN {X 0,Y 546.193,Z 244.777,A -85,B 0,C 180,E1 -3792.004,E2 -3792.004} C_VEL
LIN {X 0,Y 546.042,Z 257.703,A -85,B 0,C 180,E1 -3792.331,E2 -3792.331} C_VEL
LIN {X 0,Y 545.9,Z 269.907,A -85,B 0,C 180,E1 -3792.784,E2 -3792.784} C_VEL
LIN {X 0,Y 545.7,Z 282.195,A -85,B 0,C 180,E1 -3793.404,E2 -3793.404} C_VEL
LIN {X 0,Y 545.467,Z 292.548,A -85,B 0,C 180,E1 -3794.075,E2 -3794.075} C_VEL
LIN {X 0,Y 545.303,Z 302.17,A -85,B 0,C 180,E1 -3794.845,E2 -3794.845} C_VEL
LIN {X 0,Y 545.155,Z 311.038,A -85,B 0,C 180,E1 -3795.707,E2 -3795.707} C_VEL
LIN {X 0,Y 544.97,Z 319.273,A -85,B 0,C 180,E1 -3796.674,E2 -3796.674} C_VEL
LIN {X 0,Y 544.857,Z 327.271,A -85,B 0,C 180,E1 -3797.839,E2 -3797.839} C_VEL
LIN {X 0,Y 544.772,Z 332.682,A -85,B 0,C 180,E1 -3798.815,E2 -3798.815} C_VEL
LIN {X 0,Y 544.738,Z 337.868,A -85,B 0,C 180,E1 -3799.992,E2 -3799.992} C_VEL
LIN {X 0,Y 544.678,Z 340.489,A -85,B 0,C 180,E1 -3800.716,E2 -3800.716} C_VEL
LIN {X 0,Y 544.015,Z 342.379,A -85,B 0,C 180,E1 -3801.3,E2 -3801.3} C_VEL
LIN {X 0,Y 541.095,Z 344.845,A -85,B 0,C 180,E1 -3802.265,E2 -3802.265} C_VEL
LIN {X 0,Y 538.615,Z 346.294,A -85,B 0,C 180,E1 -3803.055,E2 -3803.055} C_VEL
LIN {X 0,Y 537.547,Z 347.072,A -85,B 0,C 180,E1 -3803.672,E2 -3803.672} C_VEL
LIN {X 0,Y 537.46,Z 347.284,A -85,B 0,C 180,E1 -3803.882,E2 -3803.882} C_VEL
LIN {X 0,Y 537.441,Z 347.7,A -85,B 0,C 180,E1 -3804.737,E2 -3804.737} C_VEL
LIN {X 0,Y 537.497,Z 347.609,A -85,B 0,C 180,E1 -3805.562,E2 -3805.562} C_VEL
LIN {X 0,Y 537.475,Z 347.08,A -85,B 0,C 180,E1 -3806.396,E2 -3806.396} C_VEL
LIN {X 0,Y 537.511,Z 346.041,A -85,B 0,C 180,E1 -3807.239,E2 -3807.239} C_VEL
LIN {X 0,Y 537.527,Z 344.459,A -85,B 0,C 180,E1 -3808.079,E2 -3808.079} C_VEL
LIN {X 0,Y 537.607,Z 341.083,A -85,B 0,C 180,E1 -3809.355,E2 -3809.355} C_VEL
LIN {X 0,Y 537.661,Z 336.255,A -85,B 0,C 180,E1 -3810.649,E2 -3810.649} C_VEL
LIN {X 0,Y 537.787,Z 330.38,A -85,B 0,C 180,E1 -3811.848,E2 -3811.848} C_VEL
LIN {X 0,Y 537.844,Z 324.389,A -85,B 0,C 180,E1 -3812.839,E2 -3812.839} C_VEL
LIN {X 0,Y 538.057,Z 316.199,A -85,B 0,C 180,E1 -3813.944,E2 -3813.944} C_VEL
LIN {X 0,Y 538.232,Z 307.101,A -85,B 0,C 180,E1 -3814.94,E2 -3814.94} C_VEL
LIN {X 0,Y 538.474,Z 296.069,A -85,B 0,C 180,E1 -3815.906,E2 -3815.906} C_VEL
LIN {X 0,Y 538.693,Z 284.829,A -85,B 0,C 180,E1 -3816.687,E2 -3816.687} C_VEL
LIN {X 0,Y 538.924,Z 272.375,A -85,B 0,C 180,E1 -3817.359,E2 -3817.359} C_VEL
LIN {X 0,Y 539.052,Z 259.273,A -85,B 0,C 180,E1 -3817.878,E2 -3817.878} C_VEL
LIN {X 0,Y 539.201,Z 246.468,A -85,B 0,C 180,E1 -3818.222,E2 -3818.222} C_VEL
LIN {X 0,Y 539.359,Z 222.061,A -85,B 0,C 180,E1 -3818.584,E2 -3818.584} C_VEL
LIN {X 0,Y 539.543,Z 145.189,A -85,B 0,C 180,E1 -3819.632,E2 -3819.632} C_VEL
LIN {X 0,Y 538.227,Z 138.018,A -85,B 0,C 180,E1 -3819.779,E2 -3819.779} C_VEL
LIN {X 0,Y 538.336,Z 124.148,A -85,B 0,C 180,E1 -3822.524,E2 -3822.524} C_VEL
LIN {X 0,Y 538.065,Z 121.464,A -85,B 0,C 180,E1 -3823.103,E2 -3823.103} C_VEL
LIN {X 0,Y 538.021,Z 121.466,A -85,B 0,C 180,E1 -3826.185,E2 -3826.185} C_VEL
LIN {X 0,Y 538.049,Z 121.461,A -85,B 0,C 180,E1 -3829.252,E2 -3829.252} C_VEL
LIN {X 0,Y 537.992,Z 121.468,A -85,B 0,C 180,E1 -3832.122,E2 -3832.122} C_VEL
LIN {X 0,Y 537.997,Z 121.466,A -85,B 0,C 180,E1 -3834.915,E2 -3834.915} C_VEL
LIN {X 0,Y 538.016,Z 121.47,A -85,B 0,C 180,E1 -3837.617,E2 -3837.617} C_VEL
LIN {X 0,Y 538.014,Z 121.463,A -85,B 0,C 180,E1 -3840.238,E2 -3840.238} C_VEL
LIN {X 0,Y 538.057,Z 121.459,A -85,B 0,C 180,E1 -3842.796,E2 -3842.796} C_VEL
LIN {X 0,Y 538.047,Z 121.467,A -85,B 0,C 180,E1 -3845.292,E2 -3845.292} C_VEL
LIN {X 0,Y 538.021,Z 121.462,A -85,B 0,C 180,E1 -3848.546,E2 -3848.546} C_VEL
LIN {X 0,Y 538.032,Z 121.465,A -85,B 0,C 180,E1 -3850.94,E2 -3850.94} C_VEL
LIN {X 0,Y 538.018,Z 121.469,A -85,B 0,C 180,E1 -3853.299,E2 -3853.299} C_VEL
LIN {X 0,Y 538.063,Z 121.459,A -85,B 0,C 180,E1 -3855.63,E2 -3855.63} C_VEL
LIN {X 0,Y 538.077,Z 121.459,A -85,B 0,C 180,E1 -3858.701,E2 -3858.701} C_VEL
LIN {X 0,Y 538.085,Z 121.454,A -85,B 0,C 180,E1 -3861.739,E2 -3861.739} C_VEL
LIN {X 0,Y 538.16,Z 121.451,A -85,B 0,C 180,E1 -3864.755,E2 -3864.755} C_VEL
LIN {X 0,Y 538.168,Z 121.443,A -85,B 0,C 180,E1 -3867.754,E2 -3867.754} C_VEL
LIN {X 0,Y 538.183,Z 121.45,A -85,B 0,C 180,E1 -3870.748,E2 -3870.748} C_VEL
LIN {X 0,Y 538.136,Z 121.453,A -85,B 0,C 180,E1 -3872.994,E2 -3872.994} C_VEL
LIN {X 0,Y 538.121,Z 121.45,A -85,B 0,C 180,E1 -3875.997,E2 -3875.997} C_VEL
LIN {X 0,Y 538.07,Z 121.459,A -85,B 0,C 180,E1 -3879.017,E2 -3879.017} C_VEL
LIN {X 0,Y 538.081,Z 121.456,A -85,B 0,C 180,E1 -3882.062,E2 -3882.062} C_VEL
LIN {X 0,Y 538.044,Z 121.46,A -85,B 0,C 180,E1 -3885.143,E2 -3885.143} C_VEL
LIN {X 0,Y 538.029,Z 121.468,A -85,B 0,C 180,E1 -3888.27,E2 -3888.27} C_VEL
LIN {X 0,Y 538.037,Z 121.464,A -85,B 0,C 180,E1 -3890.651,E2 -3890.651} C_VEL
LIN {X 0,Y 538,Z 121.467,A -85,B 0,C 180,E1 -3893.888,E2 -3893.888} C_VEL
LIN {X 0,Y 538.039,Z 121.467,A -85,B 0,C 180,E1 -3896.366,E2 -3896.366} C_VEL
LIN {X 0,Y 538.035,Z 121.46,A -85,B 0,C 180,E1 -3898.935,E2 -3898.935} C_VEL
LIN {X 0,Y 538.025,Z 121.467,A -85,B 0,C 180,E1 -3901.89,E2 -3901.89} C_VEL
LIN {X 0,Y 538.024,Z 121.463,A -85,B 0,C 180,E1 -3904.62,E2 -3904.62} C_VEL
LIN {X 0,Y 538.005,Z 121.464,A -85,B 0,C 180,E1 -3907.17,E2 -3907.17} C_VEL
LIN {X 0,Y 538.028,Z 121.467,A -85,B 0,C 180,E1 -3909.796,E2 -3909.796} C_VEL
LIN {X 0,Y 538.021,Z 121.462,A -85,B 0,C 180,E1 -3912.785,E2 -3912.785} C_VEL
LIN {X 0,Y 538.027,Z 121.469,A -85,B 0,C 180,E1 -3915.925,E2 -3915.925} C_VEL
LIN {X 0,Y 538.076,Z 121.457,A -85,B 0,C 180,E1 -3919.249,E2 -3919.249} C_VEL
LIN {X 0,Y 537.991,Z 121.468,A -85,B 0,C 180,E1 -3922.122,E2 -3922.122} C_VEL
LIN {X 0,Y 537.995,Z 121.465,A -85,B 0,C 180,E1 -3924.916,E2 -3924.916} C_VEL
LIN {X 0,Y 538.029,Z 121.469,A -85,B 0,C 180,E1 -3927.618,E2 -3927.618} C_VEL
LIN {X 0,Y 538.015,Z 121.463,A -85,B 0,C 180,E1 -3930.239,E2 -3930.239} C_VEL
LIN {X 0,Y 538.06,Z 121.458,A -85,B 0,C 180,E1 -3932.796,E2 -3932.796} C_VEL
LIN {X 0,Y 538.045,Z 121.466,A -85,B 0,C 180,E1 -3935.293,E2 -3935.293} C_VEL
LIN {X 0,Y 538.02,Z 121.462,A -85,B 0,C 180,E1 -3938.546,E2 -3938.546} C_VEL
LIN {X 0,Y 538.035,Z 121.464,A -85,B 0,C 180,E1 -3940.94,E2 -3940.94} C_VEL
LIN {X 0,Y 538.022,Z 121.47,A -85,B 0,C 180,E1 -3943.299,E2 -3943.299} C_VEL
LIN {X 0,Y 538.062,Z 121.459,A -85,B 0,C 180,E1 -3945.631,E2 -3945.631} C_VEL
LIN {X 0,Y 538.075,Z 121.458,A -85,B 0,C 180,E1 -3948.702,E2 -3948.702} C_VEL
LIN {X 0,Y 538.084,Z 121.455,A -85,B 0,C 180,E1 -3951.74,E2 -3951.74} C_VEL
LIN {X 0,Y 538.16,Z 121.45,A -85,B 0,C 180,E1 -3954.755,E2 -3954.755} C_VEL
LIN {X 0,Y 538.168,Z 121.443,A -85,B 0,C 180,E1 -3957.755,E2 -3957.755} C_VEL
LIN {X 0,Y 538.183,Z 121.449,A -85,B 0,C 180,E1 -3960.749,E2 -3960.749} C_VEL
LIN {X 0,Y 538.135,Z 121.454,A -85,B 0,C 180,E1 -3962.995,E2 -3962.995} C_VEL
LIN {X 0,Y 538.131,Z 121.448,A -85,B 0,C 180,E1 -3965.997,E2 -3965.997} C_VEL
LIN {X 0,Y 538.07,Z 121.46,A -85,B 0,C 180,E1 -3969.018,E2 -3969.018} C_VEL
LIN {X 0,Y 538.082,Z 121.456,A -85,B 0,C 180,E1 -3972.063,E2 -3972.063} C_VEL
LIN {X 0,Y 538.044,Z 121.46,A -85,B 0,C 180,E1 -3975.144,E2 -3975.144} C_VEL
LIN {X 0,Y 538.031,Z 121.466,A -85,B 0,C 180,E1 -3978.27,E2 -3978.27} C_VEL
LIN {X 0,Y 538.039,Z 121.465,A -85,B 0,C 180,E1 -3980.652,E2 -3980.652} C_VEL
LIN {X 0,Y 538.001,Z 121.467,A -85,B 0,C 180,E1 -3983.889,E2 -3983.889} C_VEL
LIN {X 0,Y 538.041,Z 121.468,A -85,B 0,C 180,E1 -3986.367,E2 -3986.367} C_VEL
LIN {X 0,Y 538.03,Z 121.461,A -85,B 0,C 180,E1 -3988.934,E2 -3988.934} C_VEL
LIN {X 0,Y 538.01,Z 121.468,A -85,B 0,C 180,E1 -3991.888,E2 -3991.888} C_VEL
LIN {X 0,Y 538.011,Z 121.465,A -85,B 0,C 180,E1 -3994.618,E2 -3994.618} C_VEL
LIN {X 0,Y 538.004,Z 121.464,A -85,B 0,C 180,E1 -3997.17,E2 -3997.17} C_VEL
LIN {X 0,Y 538.055,Z 121.463,A -85,B 0,C 180,E1 -3999.794,E2 -3999.794} C_VEL
LIN {X 0,Y 538.019,Z 121.462,A -85,B 0,C 180,E1 -4002.786,E2 -4002.786} C_VEL
LIN {X 0,Y 538.032,Z 121.461,A -85,B 0,C 180,E1 -4005.141,E2 -4005.141} C_VEL
LIN {X 0,Y 538.04,Z 121.463,A -85,B 0,C 180,E1 -4008.228,E2 -4008.228} C_VEL
LIN {X 0,Y 538.016,Z 121.464,A -85,B 0,C 180,E1 -4011.17,E2 -4011.17} C_VEL
LIN {X 0,Y 537.995,Z 121.468,A -85,B 0,C 180,E1 -4014.089,E2 -4014.089} C_VEL
LIN {X 0,Y 538.031,Z 121.46,A -85,B 0,C 180,E1 -4016.728,E2 -4016.728} C_VEL
LIN {X 0,Y 538.028,Z 121.469,A -85,B 0,C 180,E1 -4019.557,E2 -4019.557} C_VEL
LIN {X 0,Y 538.042,Z 121.464,A -85,B 0,C 180,E1 -4021.951,E2 -4021.951} C_VEL
LIN {X 0,Y 538.11,Z 121.521,A -85,B 0,C 180,E1 -4024.935,E2 -4024.935} C_VEL
LIN {X 0,Y 539.435,Z 129.548,A -85,B 0,C 180,E1 -4026.179,E2 -4026.179} C_VEL
LIN {X 0,Y 539.078,Z 147.588,A -85,B 0,C 180,E1 -4028.791,E2 -4028.791} C_VEL
LIN {X 0,Y 538.696,Z 170.634,A -85,B 0,C 180,E1 -4032.068,E2 -4032.068} C_VEL
LIN {X 0,Y 538.324,Z 191.748,A -85,B 0,C 180,E1 -4035.038,E2 -4035.038} C_VEL
LIN {X 0,Y 538.302,Z 193.234,A -85,B 0,C 180,E1 -4035.246,E2 -4035.246} C_VEL
LIN {X 0,Y 539.593,Z 202.719,A -85,B 0,C 180,E1 -4035.419,E2 -4035.419} C_VEL
LIN {X 0,Y 539.269,Z 301.754,A -85,B 0,C 180,E1 -4036.769,E2 -4036.769} C_VEL
LIN {X 0,Y 539.096,Z 314.323,A -85,B 0,C 180,E1 -4037.076,E2 -4037.076} C_VEL
LIN {X 0,Y 538.847,Z 327.87,A -85,B 0,C 180,E1 -4037.573,E2 -4037.573} C_VEL
LIN {X 0,Y 538.622,Z 339.893,A -85,B 0,C 180,E1 -4038.18,E2 -4038.18} C_VEL
LIN {X 0,Y 538.413,Z 350.979,A -85,B 0,C 180,E1 -4038.9,E2 -4038.9} C_VEL
LIN {X 0,Y 538.192,Z 361.533,A -85,B 0,C 180,E1 -4039.752,E2 -4039.752} C_VEL
LIN {X 0,Y 538.019,Z 370.163,A -85,B 0,C 180,E1 -4040.603,E2 -4040.603} C_VEL
LIN {X 0,Y 537.89,Z 378.124,A -85,B 0,C 180,E1 -4041.548,E2 -4041.548} C_VEL
LIN {X 0,Y 537.755,Z 385.897,A -85,B 0,C 180,E1 -4042.68,E2 -4042.68} C_VEL
LIN {X 0,Y 537.665,Z 393.051,A -85,B 0,C 180,E1 -4043.998,E2 -4043.998} C_VEL
LIN {X 0,Y 537.54,Z 397.808,A -85,B 0,C 180,E1 -4045.125,E2 -4045.125} C_VEL
LIN {X 0,Y 537.591,Z 401.449,A -85,B 0,C 180,E1 -4046.252,E2 -4046.252} C_VEL
LIN {X 0,Y 537.58,Z 403.324,A -85,B 0,C 180,E1 -4047.003,E2 -4047.003} C_VEL
LIN {X 0,Y 537.455,Z 405.726,A -85,B 0,C 180,E1 -4048.502,E2 -4048.502} C_VEL
LIN {X 0,Y 537.452,Z 406.337,A -85,B 0,C 180,E1 -4049.251,E2 -4049.251} C_VEL
LIN {X 0,Y 537.453,Z 406.552,A -85,B 0,C 180,E1 -4050,E2 -4050} C_VEL
LIN {X 0,Y 537.452,Z 406.333,A -85,B 0,C 180,E1 -4050.75,E2 -4050.75} C_VEL
LIN {X 0,Y 537.49,Z 404.717,A -85,B 0,C 180,E1 -4052.248,E2 -4052.248} C_VEL
LIN {X 0,Y 537.58,Z 403.309,A -85,B 0,C 180,E1 -4052.998,E2 -4052.998} C_VEL
LIN {X 0,Y 537.603,Z 400.345,A -85,B 0,C 180,E1 -4054.123,E2 -4054.123} C_VEL
LIN {X 0,Y 537.588,Z 396.328,A -85,B 0,C 180,E1 -4055.251,E2 -4055.251} C_VEL
LIN {X 0,Y 537.644,Z 390.224,A -85,B 0,C 180,E1 -4056.554,E2 -4056.554} C_VEL
LIN {X 0,Y 537.764,Z 383.401,A -85,B 0,C 180,E1 -4057.699,E2 -4057.699} C_VEL
LIN {X 0,Y 537.929,Z 375.019,A -85,B 0,C 180,E1 -4058.831,E2 -4058.831} C_VEL
LIN {X 0,Y 538.067,Z 366.409,A -85,B 0,C 180,E1 -4059.776,E2 -4059.776} C_VEL
LIN {X 0,Y 538.292,Z 355.78,A -85,B 0,C 180,E1 -4060.723,E2 -4060.723} C_VEL
LIN {X 0,Y 538.502,Z 344.539,A -85,B 0,C 180,E1 -4061.527,E2 -4061.527} C_VEL
LIN {X 0,Y 538.741,Z 333.672,A -85,B 0,C 180,E1 -4062.143,E2 -4062.143} C_VEL
LIN {X 0,Y 538.932,Z 321.678,A -85,B 0,C 180,E1 -4062.665,E2 -4062.665} C_VEL
LIN {X 0,Y 539.134,Z 307.83,A -85,B 0,C 180,E1 -4063.091,E2 -4063.091} C_VEL
LIN {X 0,Y 539.303,Z 295.192,A -85,B 0,C 180,E1 -4063.327,E2 -4063.327} C_VEL
LIN {X 0,Y 539.433,Z 201.259,A -85,B 0,C 180,E1 -4064.601,E2 -4064.601} C_VEL
LIN {X 0,Y 538.23,Z 192.608,A -85,B 0,C 180,E1 -4064.779,E2 -4064.779} C_VEL
LIN {X 0,Y 538.555,Z 173.149,A -85,B 0,C 180,E1 -4067.466,E2 -4067.466} C_VEL
LIN {X 0,Y 538.864,Z 150.586,A -85,B 0,C 180,E1 -4070.619,E2 -4070.619} C_VEL
LIN {X 0,Y 539.182,Z 130.689,A -85,B 0,C 180,E1 -4073.426,E2 -4073.426} C_VEL
LIN {X 0,Y 538.928,Z 126.025,A -85,B 0,C 180,E1 -4074.097,E2 -4074.097} C_VEL
LIN {X 0,Y 538.09,Z 121.462,A -85,B 0,C 180,E1 -4074.809,E2 -4074.809} C_VEL
LIN {X 0,Y 538.044,Z 121.467,A -85,B 0,C 180,E1 -4078.05,E2 -4078.05} C_VEL
LIN {X 0,Y 538.024,Z 121.469,A -85,B 0,C 180,E1 -4080.627,E2 -4080.627} C_VEL
LIN {X 0,Y 538.049,Z 121.459,A -85,B 0,C 180,E1 -4083.283,E2 -4083.283} C_VEL
LIN {X 0,Y 537.998,Z 121.472,A -85,B 0,C 180,E1 -4086.005,E2 -4086.005} C_VEL
LIN {X 0,Y 538.018,Z 121.464,A -85,B 0,C 180,E1 -4088.83,E2 -4088.83} C_VEL
LIN {X 0,Y 538.034,Z 121.467,A -85,B 0,C 180,E1 -4091.773,E2 -4091.773} C_VEL
LIN {X 0,Y 538.036,Z 121.461,A -85,B 0,C 180,E1 -4094.859,E2 -4094.859} C_VEL
LIN {X 0,Y 538.023,Z 121.463,A -85,B 0,C 180,E1 -4097.214,E2 -4097.214} C_VEL
LIN {X 0,Y 538.026,Z 121.463,A -85,B 0,C 180,E1 -4100.203,E2 -4100.203} C_VEL
LIN {X 0,Y 538.027,Z 121.462,A -85,B 0,C 180,E1 -4103.067,E2 -4103.067} C_VEL
LIN {X 0,Y 538.013,Z 121.467,A -85,B 0,C 180,E1 -4105.826,E2 -4105.826} C_VEL
LIN {X 0,Y 538.012,Z 121.462,A -85,B 0,C 180,E1 -4108.498,E2 -4108.498} C_VEL
LIN {X 0,Y 538.046,Z 121.464,A -85,B 0,C 180,E1 -4111.099,E2 -4111.099} C_VEL
LIN {X 0,Y 538.044,Z 121.462,A -85,B 0,C 180,E1 -4113.633,E2 -4113.633} C_VEL
LIN {X 0,Y 538.01,Z 121.464,A -85,B 0,C 180,E1 -4116.122,E2 -4116.122} C_VEL
LIN {X 0,Y 538.04,Z 121.465,A -85,B 0,C 180,E1 -4119.348,E2 -4119.348} C_VEL
LIN {X 0,Y 538.039,Z 121.46,A -85,B 0,C 180,E1 -4122.468,E2 -4122.468} C_VEL
LIN {X 0,Y 538.059,Z 121.459,A -85,B 0,C 180,E1 -4125.63,E2 -4125.63} C_VEL
LIN {X 0,Y 538.08,Z 121.462,A -85,B 0,C 180,E1 -4128.701,E2 -4128.701} C_VEL
LIN {X 0,Y 538.063,Z 121.458,A -85,B 0,C 180,E1 -4131.739,E2 -4131.739} C_VEL
LIN {X 0,Y 538.159,Z 121.454,A -85,B 0,C 180,E1 -4134.755,E2 -4134.755} C_VEL
LIN {X 0,Y 538.168,Z 121.446,A -85,B 0,C 180,E1 -4137.754,E2 -4137.754} C_VEL
LIN {X 0,Y 538.18,Z 121.449,A -85,B 0,C 180,E1 -4140.748,E2 -4140.748} C_VEL
LIN {X 0,Y 538.124,Z 121.453,A -85,B 0,C 180,E1 -4142.994,E2 -4142.994} C_VEL
LIN {X 0,Y 538.116,Z 121.457,A -85,B 0,C 180,E1 -4145.997,E2 -4145.997} C_VEL
LIN {X 0,Y 538.122,Z 121.664,A -85,B 0,C 180,E1 -4147.193,E2 -4147.193} C_VEL
LIN {X 0,Y 538.195,Z 130.411,A -85,B 0,C 180,E1 -4148.826,E2 -4148.826} C_VEL
LIN {X 0,Y 538.215,Z 138.35,A -85,B 0,C 180,E1 -4150.319,E2 -4150.319} C_VEL
LIN {X 0,Y 539.636,Z 145.326,A -85,B 0,C 180,E1 -4150.458,E2 -4150.458} C_VEL
LIN {X 0,Y 539.285,Z 245.007,A -85,B 0,C 180,E1 -4151.841,E2 -4151.841} C_VEL
LIN {X 0,Y 539.115,Z 258.135,A -85,B 0,C 180,E1 -4152.176,E2 -4152.176} C_VEL
LIN {X 0,Y 538.969,Z 270.674,A -85,B 0,C 180,E1 -4152.649,E2 -4152.649} C_VEL
LIN {X 0,Y 538.733,Z 283.107,A -85,B 0,C 180,E1 -4153.292,E2 -4153.292} C_VEL
LIN {X 0,Y 538.505,Z 294.653,A -85,B 0,C 180,E1 -4154.068,E2 -4154.068} C_VEL
LIN {X 0,Y 538.251,Z 304.957,A -85,B 0,C 180,E1 -4154.933,E2 -4154.933} C_VEL
LIN {X 0,Y 538.104,Z 314.39,A -85,B 0,C 180,E1 -4155.918,E2 -4155.918} C_VEL
LIN {X 0,Y 537.92,Z 322.083,A -85,B 0,C 180,E1 -4156.9,E2 -4156.9} C_VEL
LIN {X 0,Y 537.777,Z 329.571,A -85,B 0,C 180,E1 -4158.082,E2 -4158.082} C_VEL
LIN {X 0,Y 537.719,Z 334.639,A -85,B 0,C 180,E1 -4159.071,E2 -4159.071} C_VEL
LIN {X 0,Y 537.619,Z 339.523,A -85,B 0,C 180,E1 -4160.268,E2 -4160.268} C_VEL
LIN {X 0,Y 537.554,Z 343.222,A -85,B 0,C 180,E1 -4161.473,E2 -4161.473} C_VEL
LIN {X 0,Y 537.519,Z 345.027,A -85,B 0,C 180,E1 -4162.282,E2 -4162.282} C_VEL
LIN {X 0,Y 537.474,Z 346.413,A -85,B 0,C 180,E1 -4163.096,E2 -4163.096} C_VEL
LIN {X 0,Y 537.46,Z 347.284,A -85,B 0,C 180,E1 -4163.882,E2 -4163.882} C_VEL
LIN {X 0,Y 536.781,Z 347.742,A -85,B 0,C 180,E1 -4164.506,E2 -4164.506} C_VEL
LIN {X 0,Y 533.894,Z 347.88,A -85,B 0,C 180,E1 -4165.522,E2 -4165.522} C_VEL
LIN {X 0,Y 531.483,Z 347.485,A -85,B 0,C 180,E1 -4166.339,E2 -4166.339} C_VEL
LIN {X 0,Y 530.43,Z 346.705,A -85,B 0,C 180,E1 -4167.073,E2 -4167.073} C_VEL
LIN {X 0,Y 530.42,Z 346.517,A -85,B 0,C 180,E1 -4167.179,E2 -4167.179} C_VEL
LIN {X 0,Y 530.46,Z 344.007,A -85,B 0,C 180,E1 -4168.487,E2 -4168.487} C_VEL
LIN {X 0,Y 530.527,Z 340.206,A -85,B 0,C 180,E1 -4169.786,E2 -4169.786} C_VEL
LIN {X 0,Y 530.603,Z 334.926,A -85,B 0,C 180,E1 -4171.102,E2 -4171.102} C_VEL
LIN {X 0,Y 530.756,Z 329.329,A -85,B 0,C 180,E1 -4172.193,E2 -4172.193} C_VEL
LIN {X 0,Y 530.935,Z 320.914,A -85,B 0,C 180,E1 -4173.495,E2 -4173.495} C_VEL
LIN {X 0,Y 531.149,Z 312.198,A -85,B 0,C 180,E1 -4174.562,E2 -4174.562} C_VEL
LIN {X 0,Y 531.311,Z 303.014,A -85,B 0,C 180,E1 -4175.483,E2 -4175.483} C_VEL
LIN {X 0,Y 531.598,Z 292.532,A -85,B 0,C 180,E1 -4176.336,E2 -4176.336} C_VEL
LIN {X 0,Y 531.806,Z 281.06,A -85,B 0,C 180,E1 -4177.081,E2 -4177.081} C_VEL
LIN {X 0,Y 532.017,Z 269.376,A -85,B 0,C 180,E1 -4177.664,E2 -4177.664} C_VEL
LIN {X 0,Y 532.187,Z 256.168,A -85,B 0,C 180,E1 -4178.149,E2 -4178.149} C_VEL
LIN {X 0,Y 532.349,Z 244.06,A -85,B 0,C 180,E1 -4178.443,E2 -4178.443} C_VEL
LIN {X 0,Y 532.732,Z 146.277,A -85,B 0,C 180,E1 -4179.812,E2 -4179.812} C_VEL
LIN {X 0,Y 531.203,Z 138.288,A -85,B 0,C 180,E1 -4179.977,E2 -4179.977} C_VEL
LIN {X 0,Y 531.312,Z 124.263,A -85,B 0,C 180,E1 -4182.766,E2 -4182.766} C_VEL
LIN {X 0,Y 531.02,Z 122.342,A -85,B 0,C 180,E1 -4183.187,E2 -4183.187} C_VEL
LIN {X 0,Y 530.988,Z 122.346,A -85,B 0,C 180,E1 -4185.62,E2 -4185.62} C_VEL
LIN {X 0,Y 530.997,Z 122.337,A -85,B 0,C 180,E1 -4188.564,E2 -4188.564} C_VEL
LIN {X 0,Y 530.957,Z 122.349,A -85,B 0,C 180,E1 -4191.529,E2 -4191.529} C_VEL
LIN {X 0,Y 530.953,Z 122.342,A -85,B 0,C 180,E1 -4194.38,E2 -4194.38} C_VEL
LIN {X 0,Y 530.966,Z 122.344,A -85,B 0,C 180,E1 -4197.133,E2 -4197.133} C_VEL
LIN {X 0,Y 530.96,Z 122.345,A -85,B 0,C 180,E1 -4199.802,E2 -4199.802} C_VEL
LIN {X 0,Y 531.012,Z 122.335,A -85,B 0,C 180,E1 -4202.467,E2 -4202.467} C_VEL
LIN {X 0,Y 531.005,Z 122.339,A -85,B 0,C 180,E1 -4204.942,E2 -4204.942} C_VEL
LIN {X 0,Y 530.971,Z 122.34,A -85,B 0,C 180,E1 -4208.246,E2 -4208.246} C_VEL
LIN {X 0,Y 530.991,Z 122.339,A -85,B 0,C 180,E1 -4210.677,E2 -4210.677} C_VEL
LIN {X 0,Y 530.974,Z 122.347,A -85,B 0,C 180,E1 -4213.07,E2 -4213.07} C_VEL
LIN {X 0,Y 531.019,Z 122.338,A -85,B 0,C 180,E1 -4215.436,E2 -4215.436} C_VEL
LIN {X 0,Y 531.036,Z 122.334,A -85,B 0,C 180,E1 -4218.549,E2 -4218.549} C_VEL
LIN {X 0,Y 531.054,Z 122.331,A -85,B 0,C 180,E1 -4221.629,E2 -4221.629} C_VEL
LIN {X 0,Y 531.119,Z 122.327,A -85,B 0,C 180,E1 -4224.685,E2 -4224.685} C_VEL
LIN {X 0,Y 531.14,Z 122.319,A -85,B 0,C 180,E1 -4227.725,E2 -4227.725} C_VEL
LIN {X 0,Y 531.153,Z 122.326,A -85,B 0,C 180,E1 -4230.758,E2 -4230.758} C_VEL
LIN {X 0,Y 531.103,Z 122.328,A -85,B 0,C 180,E1 -4233.034,E2 -4233.034} C_VEL
LIN {X 0,Y 531.075,Z 122.328,A -85,B 0,C 180,E1 -4236.077,E2 -4236.077} C_VEL
LIN {X 0,Y 531.055,Z 122.335,A -85,B 0,C 180,E1 -4238.37,E2 -4238.37} C_VEL
LIN {X 0,Y 531.05,Z 122.33,A -85,B 0,C 180,E1 -4241.672,E2 -4241.672} C_VEL
LIN {X 0,Y 531.029,Z 122.335,A -85,B 0,C 180,E1 -4244.956,E2 -4244.956} C_VEL
LIN {X 0,Y 531.015,Z 122.335,A -85,B 0,C 180,E1 -4247.722,E2 -4247.722} C_VEL
LIN {X 0,Y 530.998,Z 122.338,A -85,B 0,C 180,E1 -4250.938,E2 -4250.938} C_VEL
LIN {X 0,Y 530.963,Z 122.349,A -85,B 0,C 180,E1 -4254.225,E2 -4254.225} C_VEL
LIN {X 0,Y 530.999,Z 122.339,A -85,B 0,C 180,E1 -4256.744,E2 -4256.744} C_VEL
LIN {X 0,Y 530.991,Z 122.337,A -85,B 0,C 180,E1 -4259.322,E2 -4259.322} C_VEL
LIN {X 0,Y 530.978,Z 122.348,A -85,B 0,C 180,E1 -4262.103,E2 -4262.103} C_VEL
LIN {X 0,Y 530.981,Z 122.339,A -85,B 0,C 180,E1 -4264.853,E2 -4264.853} C_VEL
LIN {X 0,Y 530.964,Z 122.343,A -85,B 0,C 180,E1 -4267.507,E2 -4267.507} C_VEL
LIN {X 0,Y 530.982,Z 122.341,A -85,B 0,C 180,E1 -4270.432,E2 -4270.432} C_VEL
LIN {X 0,Y 530.967,Z 122.342,A -85,B 0,C 180,E1 -4273.282,E2 -4273.282} C_VEL
LIN {X 0,Y 530.985,Z 122.344,A -85,B 0,C 180,E1 -4275.621,E2 -4275.621} C_VEL
LIN {X 0,Y 531.004,Z 122.336,A -85,B 0,C 180,E1 -4278.566,E2 -4278.566} C_VEL
LIN {X 0,Y 530.966,Z 122.344,A -85,B 0,C 180,E1 -4281.346,E2 -4281.346} C_VEL
LIN {X 0,Y 530.951,Z 122.343,A -85,B 0,C 180,E1 -4284.38,E2 -4284.38} C_VEL
LIN {X 0,Y 530.969,Z 122.343,A -85,B 0,C 180,E1 -4287.134,E2 -4287.134} C_VEL
LIN {X 0,Y 530.967,Z 122.345,A -85,B 0,C 180,E1 -4289.803,E2 -4289.803} C_VEL
LIN {X 0,Y 531.012,Z 122.335,A -85,B 0,C 180,E1 -4292.467,E2 -4292.467} C_VEL
LIN {X 0,Y 531.003,Z 122.338,A -85,B 0,C 180,E1 -4294.943,E2 -4294.943} C_VEL
LIN {X 0,Y 530.969,Z 122.34,A -85,B 0,C 180,E1 -4298.247,E2 -4298.247} C_VEL
LIN {X 0,Y 530.993,Z 122.338,A -85,B 0,C 180,E1 -4300.678,E2 -4300.678} C_VEL
LIN {X 0,Y 530.983,Z 122.345,A -85,B 0,C 180,E1 -4303.071,E2 -4303.071} C_VEL
LIN {X 0,Y 531.017,Z 122.339,A -85,B 0,C 180,E1 -4305.436,E2 -4305.436} C_VEL
LIN {X 0,Y 531.035,Z 122.334,A -85,B 0,C 180,E1 -4308.55,E2 -4308.55} C_VEL
LIN {X 0,Y 531.053,Z 122.331,A -85,B 0,C 180,E1 -4311.63,E2 -4311.63} C_VEL
LIN {X 0,Y 531.119,Z 122.326,A -85,B 0,C 180,E1 -4314.686,E2 -4314.686} C_VEL
LIN {X 0,Y 531.14,Z 122.319,A -85,B 0,C 180,E1 -4317.725,E2 -4317.725} C_VEL
LIN {X 0,Y 531.152,Z 122.325,A -85,B 0,C 180,E1 -4320.758,E2 -4320.758} C_VEL
LIN {X 0,Y 531.102,Z 122.329,A -85,B 0,C 180,E1 -4323.034,E2 -4323.034} C_VEL
LIN {X 0,Y 531.09,Z 122.326,A -85,B 0,C 180,E1 -4326.077,E2 -4326.077} C_VEL
LIN {X 0,Y 531.03,Z 122.335,A -85,B 0,C 180,E1 -4329.138,E2 -4329.138} C_VEL
LIN {X 0,Y 531.04,Z 122.335,A -85,B 0,C 180,E1 -4332.225,E2 -4332.225} C_VEL
LIN {X 0,Y 530.995,Z 122.337,A -85,B 0,C 180,E1 -4335.35,E2 -4335.35} C_VEL
LIN {X 0,Y 530.99,Z 122.346,A -85,B 0,C 180,E1 -4338.521,E2 -4338.521} C_VEL
LIN {X 0,Y 530.999,Z 122.338,A -85,B 0,C 180,E1 -4340.938,E2 -4340.938} C_VEL
LIN {X 0,Y 530.964,Z 122.348,A -85,B 0,C 180,E1 -4344.226,E2 -4344.226} C_VEL
LIN {X 0,Y 531.001,Z 122.339,A -85,B 0,C 180,E1 -4346.744,E2 -4346.744} C_VEL
LIN {X 0,Y 530.981,Z 122.338,A -85,B 0,C 180,E1 -4349.323,E2 -4349.323} C_VEL
LIN {X 0,Y 530.965,Z 122.349,A -85,B 0,C 180,E1 -4352.101,E2 -4352.101} C_VEL
LIN {X 0,Y 530.969,Z 122.341,A -85,B 0,C 180,E1 -4354.852,E2 -4354.852} C_VEL
LIN {X 0,Y 530.966,Z 122.342,A -85,B 0,C 180,E1 -4357.508,E2 -4357.508} C_VEL
LIN {X 0,Y 530.992,Z 122.34,A -85,B 0,C 180,E1 -4360.432,E2 -4360.432} C_VEL
LIN {X 0,Y 530.965,Z 122.343,A -85,B 0,C 180,E1 -4363.495,E2 -4363.495} C_VEL
LIN {X 0,Y 530.965,Z 122.342,A -85,B 0,C 180,E1 -4366.506,E2 -4366.506} C_VEL
LIN {X 0,Y 530.988,Z 122.343,A -85,B 0,C 180,E1 -4369.568,E2 -4369.568} C_VEL
LIN {X 0,Y 530.969,Z 122.34,A -85,B 0,C 180,E1 -4372.577,E2 -4372.577} C_VEL
LIN {X 0,Y 530.983,Z 122.342,A -85,B 0,C 180,E1 -4375.31,E2 -4375.31} C_VEL
LIN {X 0,Y 530.968,Z 122.344,A -85,B 0,C 180,E1 -4378.032,E2 -4378.032} C_VEL
LIN {X 0,Y 530.99,Z 122.339,A -85,B 0,C 180,E1 -4380.875,E2 -4380.875} C_VEL
LIN {X 0,Y 531.004,Z 122.343,A -85,B 0,C 180,E1 -4383.257,E2 -4383.257} C_VEL
LIN {X 0,Y 531.053,Z 122.423,A -85,B 0,C 180,E1 -4384.762,E2 -4384.762} C_VEL
LIN {X 0,Y 532.51,Z 130.643,A -85,B 0,C 180,E1 -4386.057,E2 -4386.057} C_VEL
LIN {X 0,Y 532.12,Z 148.646,A -85,B 0,C 180,E1 -4388.703,E2 -4388.703} C_VEL
LIN {X 0,Y 531.683,Z 170.67,A -85,B 0,C 180,E1 -4391.877,E2 -4391.877} C_VEL
LIN {X 0,Y 531.304,Z 192.101,A -85,B 0,C 180,E1 -4394.936,E2 -4394.936} C_VEL
LIN {X 0,Y 531.295,Z 193.212,A -85,B 0,C 180,E1 -4395.055,E2 -4395.055} C_VEL
LIN {X 0,Y 532.727,Z 204.53,A -85,B 0,C 180,E1 -4395.257,E2 -4395.257} C_VEL
LIN {X 0,Y 532.354,Z 300.922,A -85,B 0,C 180,E1 -4396.594,E2 -4396.594} C_VEL
LIN {X 0,Y 532.175,Z 312.9,A -85,B 0,C 180,E1 -4396.881,E2 -4396.881} C_VEL
LIN {X 0,Y 531.944,Z 325.017,A -85,B 0,C 180,E1 -4397.312,E2 -4397.312} C_VEL
LIN {X 0,Y 531.692,Z 337.425,A -85,B 0,C 180,E1 -4397.913,E2 -4397.913} C_VEL
LIN {X 0,Y 531.452,Z 349.182,A -85,B 0,C 180,E1 -4398.656,E2 -4398.656} C_VEL
LIN {X 0,Y 531.209,Z 359.982,A -85,B 0,C 180,E1 -4399.519,E2 -4399.519} C_VEL
LIN {X 0,Y 530.973,Z 369.709,A -85,B 0,C 180,E1 -4400.477,E2 -4400.477} C_VEL
LIN {X 0,Y 530.799,Z 377.684,A -85,B 0,C 180,E1 -4401.434,E2 -4401.434} C_VEL
LIN {X 0,Y 530.665,Z 385.477,A -85,B 0,C 180,E1 -4402.581,E2 -4402.581} C_VEL
LIN {X 0,Y 530.559,Z 392.643,A -85,B 0,C 180,E1 -4403.917,E2 -4403.917} C_VEL
LIN {X 0,Y 530.459,Z 397.409,A -85,B 0,C 180,E1 -4405.06,E2 -4405.06} C_VEL
LIN {X 0,Y 530.516,Z 401.057,A -85,B 0,C 180,E1 -4406.202,E2 -4406.202} C_VEL
LIN {X 0,Y 530.512,Z 402.937,A -85,B 0,C 180,E1 -4406.963,E2 -4406.963} C_VEL
LIN {X 0,Y 530.365,Z 405.34,A -85,B 0,C 180,E1 -4408.482,E2 -4408.482} C_VEL
LIN {X 0,Y 530.362,Z 405.951,A -85,B 0,C 180,E1 -4409.241,E2 -4409.241} C_VEL
LIN {X 0,Y 530.364,Z 406.165,A -85,B 0,C 180,E1 -4410,E2 -4410} C_VEL
LIN {X 0,Y 530.362,Z 405.943,A -85,B 0,C 180,E1 -4410.76,E2 -4410.76} C_VEL
LIN {X 0,Y 530.412,Z 404.32,A -85,B 0,C 180,E1 -4412.278,E2 -4412.278} C_VEL
LIN {X 0,Y 530.512,Z 402.906,A -85,B 0,C 180,E1 -4413.038,E2 -4413.038} C_VEL
LIN {X 0,Y 530.522,Z 399.931,A -85,B 0,C 180,E1 -4414.179,E2 -4414.179} C_VEL
LIN {X 0,Y 530.522,Z 395.901,A -85,B 0,C 180,E1 -4415.321,E2 -4415.321} C_VEL
LIN {X 0,Y 530.543,Z 390.381,A -85,B 0,C 180,E1 -4416.529,E2 -4416.529} C_VEL
LIN {X 0,Y 530.673,Z 384.181,A -85,B 0,C 180,E1 -4417.611,E2 -4417.611} C_VEL
LIN {X 0,Y 530.829,Z 376.04,A -85,B 0,C 180,E1 -4418.758,E2 -4418.758} C_VEL
LIN {X 0,Y 530.982,Z 367.729,A -85,B 0,C 180,E1 -4419.716,E2 -4419.716} C_VEL
LIN {X 0,Y 531.223,Z 357.584,A -85,B 0,C 180,E1 -4420.674,E2 -4420.674} C_VEL
LIN {X 0,Y 531.445,Z 346.008,A -85,B 0,C 180,E1 -4421.544,E2 -4421.544} C_VEL
LIN {X 0,Y 531.707,Z 334.834,A -85,B 0,C 180,E1 -4422.21,E2 -4422.21} C_VEL
LIN {X 0,Y 531.964,Z 322.249,A -85,B 0,C 180,E1 -4422.785,E2 -4422.785} C_VEL
LIN {X 0,Y 532.201,Z 308.809,A -85,B 0,C 180,E1 -4423.216,E2 -4423.216} C_VEL
LIN {X 0,Y 532.369,Z 295.686,A -85,B 0,C 180,E1 -4423.479,E2 -4423.479} C_VEL
LIN {X 0,Y 532.559,Z 202.085,A -85,B 0,C 180,E1 -4424.776,E2 -4424.776} C_VEL
LIN {X 0,Y 531.203,Z 192.281,A -85,B 0,C 180,E1 -4424.961,E2 -4424.961} C_VEL
LIN {X 0,Y 531.548,Z 171.798,A -85,B 0,C 180,E1 -4427.83,E2 -4427.83} C_VEL
LIN {X 0,Y 531.926,Z 148.671,A -85,B 0,C 180,E1 -4431.103,E2 -4431.103} C_VEL
LIN {X 0,Y 532.228,Z 130.136,A -85,B 0,C 180,E1 -4433.75,E2 -4433.75} C_VEL
LIN {X 0,Y 531.075,Z 122.334,A -85,B 0,C 180,E1 -4434.95,E2 -4434.95} C_VEL
LIN {X 0,Y 531.017,Z 122.339,A -85,B 0,C 180,E1 -4437.596,E2 -4437.596} C_VEL
LIN {X 0,Y 530.978,Z 122.347,A -85,B 0,C 180,E1 -4440.645,E2 -4440.645} C_VEL
LIN {X 0,Y 530.991,Z 122.342,A -85,B 0,C 180,E1 -4443.773,E2 -4443.773} C_VEL
LIN {X 0,Y 530.959,Z 122.346,A -85,B 0,C 180,E1 -4446.558,E2 -4446.558} C_VEL
LIN {X 0,Y 530.991,Z 122.34,A -85,B 0,C 180,E1 -4449.443,E2 -4449.443} C_VEL
LIN {X 0,Y 530.981,Z 122.342,A -85,B 0,C 180,E1 -4452.457,E2 -4452.457} C_VEL
LIN {X 0,Y 530.992,Z 122.344,A -85,B 0,C 180,E1 -4455.621,E2 -4455.621} C_VEL
LIN {X 0,Y 530.998,Z 122.336,A -85,B 0,C 180,E1 -4458.564,E2 -4458.564} C_VEL
LIN {X 0,Y 530.961,Z 122.346,A -85,B 0,C 180,E1 -4461.529,E2 -4461.529} C_VEL
LIN {X 0,Y 530.957,Z 122.342,A -85,B 0,C 180,E1 -4464.38,E2 -4464.38} C_VEL
LIN {X 0,Y 530.97,Z 122.343,A -85,B 0,C 180,E1 -4467.133,E2 -4467.133} C_VEL
LIN {X 0,Y 530.965,Z 122.345,A -85,B 0,C 180,E1 -4469.802,E2 -4469.802} C_VEL
LIN {X 0,Y 531.015,Z 122.335,A -85,B 0,C 180,E1 -4472.468,E2 -4472.468} C_VEL
LIN {X 0,Y 531.002,Z 122.339,A -85,B 0,C 180,E1 -4474.942,E2 -4474.942} C_VEL
LIN {X 0,Y 530.975,Z 122.34,A -85,B 0,C 180,E1 -4478.247,E2 -4478.247} C_VEL
LIN {X 0,Y 530.986,Z 122.341,A -85,B 0,C 180,E1 -4480.677,E2 -4480.677} C_VEL
LIN {X 0,Y 530.967,Z 122.349,A -85,B 0,C 180,E1 -4483.07,E2 -4483.07} C_VEL
LIN {X 0,Y 531.017,Z 122.338,A -85,B 0,C 180,E1 -4485.436,E2 -4485.436} C_VEL
LIN {X 0,Y 531.038,Z 122.337,A -85,B 0,C 180,E1 -4488.549,E2 -4488.549} C_VEL
LIN {X 0,Y 531.038,Z 122.334,A -85,B 0,C 180,E1 -4491.629,E2 -4491.629} C_VEL
LIN {X 0,Y 531.118,Z 122.332,A -85,B 0,C 180,E1 -4494.685,E2 -4494.685} C_VEL
LIN {X 0,Y 531.14,Z 122.322,A -85,B 0,C 180,E1 -4497.725,E2 -4497.725} C_VEL
LIN {X 0,Y 531.15,Z 122.324,A -85,B 0,C 180,E1 -4500.758,E2 -4500.758} C_VEL
LIN {X 0,Y 531.091,Z 122.329,A -85,B 0,C 180,E1 -4503.034,E2 -4503.034} C_VEL
LIN {X 0,Y 531.072,Z 122.336,A -85,B 0,C 180,E1 -4506.077,E2 -4506.077} C_VEL
LIN {X 0,Y 531.083,Z 122.357,A -85,B 0,C 180,E1 -4507.058,E2 -4507.058} C_VEL
LIN {X 0,Y 531.245,Z 129.385,A -85,B 0,C 180,E1 -4508.367,E2 -4508.367} C_VEL
LIN {X 0,Y 531.216,Z 138.691,A -85,B 0,C 180,E1 -4510.12,E2 -4510.12} C_VEL
LIN {X 0,Y 532.838,Z 146.655,A -85,B 0,C 180,E1 -4510.281,E2 -4510.281} C_VEL
LIN {X 0,Y 532.343,Z 245.949,A -85,B 0,C 180,E1 -4511.688,E2 -4511.688} C_VEL
LIN {X 0,Y 532.207,Z 259.183,A -85,B 0,C 180,E1 -4512.037,E2 -4512.037} C_VEL
LIN {X 0,Y 532.024,Z 271.239,A -85,B 0,C 180,E1 -4512.502,E2 -4512.502} C_VEL
LIN {X 0,Y 531.799,Z 282.41,A -85,B 0,C 180,E1 -4513.08,E2 -4513.08} C_VEL
LIN {X 0,Y 531.523,Z 294.197,A -85,B 0,C 180,E1 -4513.866,E2 -4513.866} C_VEL
LIN {X 0,Y 531.34,Z 303.848,A -85,B 0,C 180,E1 -4514.67,E2 -4514.67} C_VEL
LIN {X 0,Y 531.153,Z 312.469,A -85,B 0,C 180,E1 -4515.541,E2 -4515.541} C_VEL
LIN {X 0,Y 530.926,Z 320.6,A -85,B 0,C 180,E1 -4516.535,E2 -4516.535} C_VEL
LIN {X 0,Y 530.757,Z 328.471,A -85,B 0,C 180,E1 -4517.731,E2 -4517.731} C_VEL
LIN {X 0,Y 530.679,Z 334.754,A -85,B 0,C 180,E1 -4518.933,E2 -4518.933} C_VEL
LIN {X 0,Y 530.577,Z 339.702,A -85,B 0,C 180,E1 -4520.145,E2 -4520.145} C_VEL
LIN {X 0,Y 530.503,Z 343.453,A -85,B 0,C 180,E1 -4521.365,E2 -4521.365} C_VEL
LIN {X 0,Y 530.418,Z 346.096,A -85,B 0,C 180,E1 -4522.597,E2 -4522.597} C_VEL
LIN {X 0,Y 530.376,Z 347.697,A -85,B 0,C 180,E1 -4523.891,E2 -4523.891} C_VEL
LIN {X 0,Y 530.364,Z 348.143,A -85,B 0,C 180,E1 -4525.09,E2 -4525.09} C_VEL
LIN {X 0,Y 530.412,Z 347.85,A -85,B 0,C 180,E1 -4525.928,E2 -4525.928} C_VEL
LIN {X 0,Y 530.42,Z 346.517,A -85,B 0,C 180,E1 -4527.179,E2 -4527.179} C_VEL
LIN {X 0,Y 529.801,Z 345.547,A -85,B 0,C 180,E1 -4527.805,E2 -4527.805} C_VEL
LIN {X 0,Y 526.964,Z 343.477,A -85,B 0,C 180,E1 -4528.812,E2 -4528.812} C_VEL
LIN {X 0,Y 524.561,Z 341.291,A -85,B 0,C 180,E1 -4529.607,E2 -4529.607} C_VEL
LIN {X 0,Y 523.555,Z 339.275,A -85,B 0,C 180,E1 -4530.208,E2 -4530.208} C_VEL
LIN {X 0,Y 523.489,Z 338.508,A -85,B 0,C 180,E1 -4530.408,E2 -4530.408} C_VEL
LIN {X 0,Y 523.633,Z 333.497,A -85,B 0,C 180,E1 -4531.563,E2 -4531.563} C_VEL
LIN {X 0,Y 523.793,Z 327.34,A -85,B 0,C 180,E1 -4532.687,E2 -4532.687} C_VEL
LIN {X 0,Y 523.925,Z 320.339,A -85,B 0,C 180,E1 -4533.728,E2 -4533.728} C_VEL
LIN {X 0,Y 524.125,Z 312.036,A -85,B 0,C 180,E1 -4534.742,E2 -4534.742} C_VEL
LIN {X 0,Y 524.366,Z 301.551,A -85,B 0,C 180,E1 -4535.781,E2 -4535.781} C_VEL
LIN {X 0,Y 524.663,Z 291.619,A -85,B 0,C 180,E1 -4536.573,E2 -4536.573} C_VEL
LIN {X 0,Y 524.889,Z 280.35,A -85,B 0,C 180,E1 -4537.291,E2 -4537.291} C_VEL
LIN {X 0,Y 525.141,Z 267.529,A -85,B 0,C 180,E1 -4537.918,E2 -4537.918} C_VEL
LIN {X 0,Y 525.323,Z 254.924,A -85,B 0,C 180,E1 -4538.362,E2 -4538.362} C_VEL
LIN {X 0,Y 525.455,Z 241.787,A -85,B 0,C 180,E1 -4538.657,E2 -4538.657} C_VEL
LIN {X 0,Y 525.823,Z 146.771,A -85,B 0,C 180,E1 -4540.008,E2 -4540.008} C_VEL
LIN {X 0,Y 524.219,Z 138.56,A -85,B 0,C 180,E1 -4540.183,E2 -4540.183} C_VEL
LIN {X 0,Y 524.279,Z 125.05,A -85,B 0,C 180,E1 -4542.881,E2 -4542.881} C_VEL
LIN {X 0,Y 523.989,Z 123.218,A -85,B 0,C 180,E1 -4543.292,E2 -4543.292} C_VEL
LIN {X 0,Y 523.928,Z 123.22,A -85,B 0,C 180,E1 -4546.415,E2 -4546.415} C_VEL
LIN {X 0,Y 523.941,Z 123.216,A -85,B 0,C 180,E1 -4548.908,E2 -4548.908} C_VEL
LIN {X 0,Y 523.915,Z 123.224,A -85,B 0,C 180,E1 -4551.898,E2 -4551.898} C_VEL
LIN {X 0,Y 523.923,Z 123.219,A -85,B 0,C 180,E1 -4554.911,E2 -4554.911} C_VEL
LIN {X 0,Y 523.934,Z 123.223,A -85,B 0,C 180,E1 -4557.679,E2 -4557.679} C_VEL
LIN {X 0,Y 523.953,Z 123.215,A -85,B 0,C 180,E1 -4560.676,E2 -4560.676} C_VEL
LIN {X 0,Y 523.973,Z 123.215,A -85,B 0,C 180,E1 -4563.728,E2 -4563.728} C_VEL
LIN {X 0,Y 523.925,Z 123.217,A -85,B 0,C 180,E1 -4566.27,E2 -4566.27} C_VEL
LIN {X 0,Y 523.945,Z 123.217,A -85,B 0,C 180,E1 -4568.766,E2 -4568.766} C_VEL
LIN {X 0,Y 523.947,Z 123.224,A -85,B 0,C 180,E1 -4571.22,E2 -4571.22} C_VEL
LIN {X 0,Y 523.931,Z 123.219,A -85,B 0,C 180,E1 -4573.638,E2 -4573.638} C_VEL
LIN {X 0,Y 523.938,Z 123.216,A -85,B 0,C 180,E1 -4576.028,E2 -4576.028} C_VEL
LIN {X 0,Y 524.012,Z 123.208,A -85,B 0,C 180,E1 -4578.394,E2 -4578.394} C_VEL
LIN {X 0,Y 524.002,Z 123.21,A -85,B 0,C 180,E1 -4581.516,E2 -4581.516} C_VEL
LIN {X 0,Y 524.08,Z 123.203,A -85,B 0,C 180,E1 -4584.613,E2 -4584.613} C_VEL
LIN {X 0,Y 524.112,Z 123.194,A -85,B 0,C 180,E1 -4587.694,E2 -4587.694} C_VEL
LIN {X 0,Y 524.123,Z 123.202,A -85,B 0,C 180,E1 -4590.768,E2 -4590.768} C_VEL
LIN {X 0,Y 524.069,Z 123.204,A -85,B 0,C 180,E1 -4593.075,E2 -4593.075} C_VEL
LIN {X 0,Y 524.037,Z 123.206,A -85,B 0,C 180,E1 -4596.159,E2 -4596.159} C_VEL
LIN {X 0,Y 524.003,Z 123.215,A -85,B 0,C 180,E1 -4598.484,E2 -4598.484} C_VEL
LIN {X 0,Y 524.001,Z 123.208,A -85,B 0,C 180,E1 -4601.739,E2 -4601.739} C_VEL
LIN {X 0,Y 523.992,Z 123.211,A -85,B 0,C 180,E1 -4605.053,E2 -4605.053} C_VEL
LIN {X 0,Y 523.962,Z 123.216,A -85,B 0,C 180,E1 -4607.969,E2 -4607.969} C_VEL
LIN {X 0,Y 523.97,Z 123.221,A -85,B 0,C 180,E1 -4610.41,E2 -4610.41} C_VEL
LIN {X 0,Y 523.908,Z 123.221,A -85,B 0,C 180,E1 -4612.893,E2 -4612.893} C_VEL
LIN {X 0,Y 523.982,Z 123.216,A -85,B 0,C 180,E1 -4616.02,E2 -4616.02} C_VEL
LIN {X 0,Y 523.94,Z 123.216,A -85,B 0,C 180,E1 -4618.874,E2 -4618.874} C_VEL
LIN {X 0,Y 523.931,Z 123.218,A -85,B 0,C 180,E1 -4621.543,E2 -4621.543} C_VEL
LIN {X 0,Y 523.938,Z 123.222,A -85,B 0,C 180,E1 -4624.289,E2 -4624.289} C_VEL
LIN {X 0,Y 523.909,Z 123.22,A -85,B 0,C 180,E1 -4627.132,E2 -4627.132} C_VEL
LIN {X 0,Y 523.934,Z 123.223,A -85,B 0,C 180,E1 -4630.13,E2 -4630.13} C_VEL
LIN {X 0,Y 523.937,Z 123.218,A -85,B 0,C 180,E1 -4632.459,E2 -4632.459} C_VEL
LIN {X 0,Y 523.953,Z 123.216,A -85,B 0,C 180,E1 -4635.309,E2 -4635.309} C_VEL
LIN {X 0,Y 523.97,Z 123.212,A -85,B 0,C 180,E1 -4638.688,E2 -4638.688} C_VEL
LIN {X 0,Y 523.922,Z 123.219,A -85,B 0,C 180,E1 -4641.079,E2 -4641.079} C_VEL
LIN {X 0,Y 523.897,Z 123.227,A -85,B 0,C 180,E1 -4643.825,E2 -4643.825} C_VEL
LIN {X 0,Y 523.939,Z 123.216,A -85,B 0,C 180,E1 -4646.636,E2 -4646.636} C_VEL
LIN {X 0,Y 523.954,Z 123.22,A -85,B 0,C 180,E1 -4649.356,E2 -4649.356} C_VEL
LIN {X 0,Y 523.975,Z 123.211,A -85,B 0,C 180,E1 -4652.281,E2 -4652.281} C_VEL
LIN {X 0,Y 523.95,Z 123.215,A -85,B 0,C 180,E1 -4654.582,E2 -4654.582} C_VEL
LIN {X 0,Y 523.909,Z 123.225,A -85,B 0,C 180,E1 -4657.107,E2 -4657.107} C_VEL
LIN {X 0,Y 523.976,Z 123.213,A -85,B 0,C 180,E1 -4659.866,E2 -4659.866} C_VEL
LIN {X 0,Y 523.964,Z 123.216,A -85,B 0,C 180,E1 -4662.837,E2 -4662.837} C_VEL
LIN {X 0,Y 523.975,Z 123.22,A -85,B 0,C 180,E1 -4665.236,E2 -4665.236} C_VEL
LIN {X 0,Y 524.01,Z 123.208,A -85,B 0,C 180,E1 -4668.394,E2 -4668.394} C_VEL
LIN {X 0,Y 524.001,Z 123.211,A -85,B 0,C 180,E1 -4671.516,E2 -4671.516} C_VEL
LIN {X 0,Y 524.08,Z 123.202,A -85,B 0,C 180,E1 -4674.614,E2 -4674.614} C_VEL
LIN {X 0,Y 524.112,Z 123.195,A -85,B 0,C 180,E1 -4677.695,E2 -4677.695} C_VEL
LIN {X 0,Y 524.122,Z 123.201,A -85,B 0,C 180,E1 -4680.769,E2 -4680.769} C_VEL
LIN {X 0,Y 524.069,Z 123.205,A -85,B 0,C 180,E1 -4683.075,E2 -4683.075} C_VEL
LIN {X 0,Y 524.051,Z 123.203,A -85,B 0,C 180,E1 -4686.159,E2 -4686.159} C_VEL
LIN {X 0,Y 523.998,Z 123.21,A -85,B 0,C 180,E1 -4689.262,E2 -4689.262} C_VEL
LIN {X 0,Y 524.002,Z 123.208,A -85,B 0,C 180,E1 -4691.74,E2 -4691.74} C_VEL
LIN {X 0,Y 523.993,Z 123.211,A -85,B 0,C 180,E1 -4695.053,E2 -4695.053} C_VEL
LIN {X 0,Y 523.963,Z 123.215,A -85,B 0,C 180,E1 -4697.969,E2 -4697.969} C_VEL
LIN {X 0,Y 523.971,Z 123.221,A -85,B 0,C 180,E1 -4700.41,E2 -4700.41} C_VEL
LIN {X 0,Y 523.909,Z 123.222,A -85,B 0,C 180,E1 -4702.894,E2 -4702.894} C_VEL
LIN {X 0,Y 523.983,Z 123.215,A -85,B 0,C 180,E1 -4706.02,E2 -4706.02} C_VEL
LIN {X 0,Y 523.938,Z 123.217,A -85,B 0,C 180,E1 -4708.875,E2 -4708.875} C_VEL
LIN {X 0,Y 523.92,Z 123.219,A -85,B 0,C 180,E1 -4711.545,E2 -4711.545} C_VEL
LIN {X 0,Y 523.932,Z 123.223,A -85,B 0,C 180,E1 -4714.291,E2 -4714.291} C_VEL
LIN {X 0,Y 523.907,Z 123.22,A -85,B 0,C 180,E1 -4717.133,E2 -4717.133} C_VEL
LIN {X 0,Y 523.969,Z 123.219,A -85,B 0,C 180,E1 -4720.134,E2 -4720.134} C_VEL
LIN {X 0,Y 523.922,Z 123.218,A -85,B 0,C 180,E1 -4723.167,E2 -4723.167} C_VEL
LIN {X 0,Y 523.942,Z 123.223,A -85,B 0,C 180,E1 -4725.773,E2 -4725.773} C_VEL
LIN {X 0,Y 523.945,Z 123.215,A -85,B 0,C 180,E1 -4728.909,E2 -4728.909} C_VEL
LIN {X 0,Y 523.918,Z 123.225,A -85,B 0,C 180,E1 -4731.899,E2 -4731.899} C_VEL
LIN {X 0,Y 523.925,Z 123.218,A -85,B 0,C 180,E1 -4734.912,E2 -4734.912} C_VEL
LIN {X 0,Y 523.936,Z 123.225,A -85,B 0,C 180,E1 -4737.68,E2 -4737.68} C_VEL
LIN {X 0,Y 523.956,Z 123.215,A -85,B 0,C 180,E1 -4740.677,E2 -4740.677} C_VEL
LIN {X 0,Y 523.976,Z 123.22,A -85,B 0,C 180,E1 -4743.729,E2 -4743.729} C_VEL
LIN {X 0,Y 524.006,Z 123.316,A -85,B 0,C 180,E1 -4744.584,E2 -4744.584} C_VEL
LIN {X 0,Y 525.555,Z 131.71,A -85,B 0,C 180,E1 -4745.93,E2 -4745.93} C_VEL
LIN {X 0,Y 525.218,Z 146.949,A -85,B 0,C 180,E1 -4748.203,E2 -4748.203} C_VEL
LIN {X 0,Y 524.824,Z 166.352,A -85,B 0,C 180,E1 -4751.051,E2 -4751.051} C_VEL
LIN {X 0,Y 524.376,Z 185.677,A -85,B 0,C 180,E1 -4753.853,E2 -4753.853} C_VEL
LIN {X 0,Y 524.289,Z 192.753,A -85,B 0,C 180,E1 -4754.849,E2 -4754.849} C_VEL
LIN {X 0,Y 525.854,Z 204.347,A -85,B 0,C 180,E1 -4755.063,E2 -4755.063} C_VEL
LIN {X 0,Y 525.428,Z 301.324,A -85,B 0,C 180,E1 -4756.439,E2 -4756.439} C_VEL
LIN {X 0,Y 525.206,Z 313.771,A -85,B 0,C 180,E1 -4756.753,E2 -4756.753} C_VEL
LIN {X 0,Y 524.932,Z 326.69,A -85,B 0,C 180,E1 -4757.238,E2 -4757.238} C_VEL
LIN {X 0,Y 524.66,Z 338.776,A -85,B 0,C 180,E1 -4757.856,E2 -4757.856} C_VEL
LIN {X 0,Y 524.412,Z 349.986,A -85,B 0,C 180,E1 -4758.599,E2 -4758.599} C_VEL
LIN {X 0,Y 524.167,Z 360.588,A -85,B 0,C 180,E1 -4759.474,E2 -4759.474} C_VEL
LIN {X 0,Y 523.922,Z 369.254,A -85,B 0,C 180,E1 -4760.347,E2 -4760.347} C_VEL
LIN {X 0,Y 523.722,Z 377.245,A -85,B 0,C 180,E1 -4761.317,E2 -4761.317} C_VEL
LIN {X 0,Y 523.576,Z 385.057,A -85,B 0,C 180,E1 -4762.48,E2 -4762.48} C_VEL
LIN {X 0,Y 523.457,Z 392.234,A -85,B 0,C 180,E1 -4763.834,E2 -4763.834} C_VEL
LIN {X 0,Y 523.383,Z 397.011,A -85,B 0,C 180,E1 -4764.993,E2 -4764.993} C_VEL
LIN {X 0,Y 523.443,Z 400.666,A -85,B 0,C 180,E1 -4766.151,E2 -4766.151} C_VEL
LIN {X 0,Y 523.417,Z 402.548,A -85,B 0,C 180,E1 -4766.922,E2 -4766.922} C_VEL
LIN {X 0,Y 523.338,Z 403.954,A -85,B 0,C 180,E1 -4767.691,E2 -4767.691} C_VEL
LIN {X 0,Y 523.272,Z 405.565,A -85,B 0,C 180,E1 -4769.231,E2 -4769.231} C_VEL
LIN {X 0,Y 523.275,Z 405.778,A -85,B 0,C 180,E1 -4770,E2 -4770} C_VEL
LIN {X 0,Y 523.272,Z 405.554,A -85,B 0,C 180,E1 -4770.77,E2 -4770.77} C_VEL
LIN {X 0,Y 523.338,Z 403.922,A -85,B 0,C 180,E1 -4772.309,E2 -4772.309} C_VEL
LIN {X 0,Y 523.417,Z 402.502,A -85,B 0,C 180,E1 -4773.079,E2 -4773.079} C_VEL
LIN {X 0,Y 523.423,Z 399.516,A -85,B 0,C 180,E1 -4774.235,E2 -4774.235} C_VEL
LIN {X 0,Y 523.456,Z 395.475,A -85,B 0,C 180,E1 -4775.393,E2 -4775.393} C_VEL
LIN {X 0,Y 523.492,Z 389.342,A -85,B 0,C 180,E1 -4776.73,E2 -4776.73} C_VEL
LIN {X 0,Y 523.64,Z 382.467,A -85,B 0,C 180,E1 -4777.908,E2 -4777.908} C_VEL
LIN {X 0,Y 523.791,Z 374.033,A -85,B 0,C 180,E1 -4779.071,E2 -4779.071} C_VEL
LIN {X 0,Y 523.969,Z 365.36,A -85,B 0,C 180,E1 -4780.042,E2 -4780.042} C_VEL
LIN {X 0,Y 524.265,Z 354.668,A -85,B 0,C 180,E1 -4781.013,E2 -4781.013} C_VEL
LIN {X 0,Y 524.507,Z 343.202,A -85,B 0,C 180,E1 -4781.849,E2 -4781.849} C_VEL
LIN {X 0,Y 524.77,Z 331.353,A -85,B 0,C 180,E1 -4782.521,E2 -4782.521} C_VEL
LIN {X 0,Y 525.031,Z 318.895,A -85,B 0,C 180,E1 -4783.055,E2 -4783.055} C_VEL
LIN {X 0,Y 525.254,Z 306.113,A -85,B 0,C 180,E1 -4783.443,E2 -4783.443} C_VEL
LIN {X 0,Y 525.487,Z 291.035,A -85,B 0,C 180,E1 -4783.708,E2 -4783.708} C_VEL
LIN {X 0,Y 525.771,Z 203.315,A -85,B 0,C 180,E1 -4784.947,E2 -4784.947} C_VEL
LIN {X 0,Y 524.191,Z 191.787,A -85,B 0,C 180,E1 -4785.172,E2 -4785.172} C_VEL
LIN {X 0,Y 524.549,Z 170.97,A -85,B 0,C 180,E1 -4788.13,E2 -4788.13} C_VEL
LIN {X 0,Y 524.954,Z 149.599,A -85,B 0,C 180,E1 -4791.191,E2 -4791.191} C_VEL
LIN {X 0,Y 525.257,Z 131.118,A -85,B 0,C 180,E1 -4793.865,E2 -4793.865} C_VEL
LIN {X 0,Y 524.038,Z 123.21,A -85,B 0,C 180,E1 -4795.096,E2 -4795.096} C_VEL
LIN {X 0,Y 523.972,Z 123.22,A -85,B 0,C 180,E1 -4797.999,E2 -4797.999} C_VEL
LIN {X 0,Y 523.948,Z 123.22,A -85,B 0,C 180,E1 -4800.855,E2 -4800.855} C_VEL
LIN {X 0,Y 523.963,Z 123.217,A -85,B 0,C 180,E1 -4803.734,E2 -4803.734} C_VEL
LIN {X 0,Y 523.907,Z 123.226,A -85,B 0,C 180,E1 -4806.401,E2 -4806.401} C_VEL
LIN {X 0,Y 523.925,Z 123.219,A -85,B 0,C 180,E1 -4809.085,E2 -4809.085} C_VEL
LIN {X 0,Y 523.955,Z 123.222,A -85,B 0,C 180,E1 -4812.119,E2 -4812.119} C_VEL
LIN {X 0,Y 523.96,Z 123.216,A -85,B 0,C 180,E1 -4815.309,E2 -4815.309} C_VEL
LIN {X 0,Y 523.96,Z 123.212,A -85,B 0,C 180,E1 -4818.69,E2 -4818.69} C_VEL
LIN {X 0,Y 523.921,Z 123.218,A -85,B 0,C 180,E1 -4821.081,E2 -4821.081} C_VEL
LIN {X 0,Y 523.904,Z 123.226,A -85,B 0,C 180,E1 -4823.825,E2 -4823.825} C_VEL
LIN {X 0,Y 523.916,Z 123.218,A -85,B 0,C 180,E1 -4826.633,E2 -4826.633} C_VEL
LIN {X 0,Y 523.952,Z 123.22,A -85,B 0,C 180,E1 -4829.355,E2 -4829.355} C_VEL
LIN {X 0,Y 523.979,Z 123.212,A -85,B 0,C 180,E1 -4832.282,E2 -4832.282} C_VEL
